LIN {X 0,Y 135.592,Z 571.454,A -85,B 0,C 180,E1 -25460.01,E2 -25460.01} C_VEL
LIN {X 0,Y 130.179,Z 578.331,A -85,B 0,C 180,E1 -25465.363,E2 -25465.363} C_VEL
LIN {X 0,Y 125.633,Z 584.379,A -85,B 0,C 180,E1 -25471.45,E2 -25471.45} C_VEL
LIN {X 0,Y 122.158,Z 589.423,A -85,B 0,C 180,E1 -25478.277,E2 -25478.277} C_VEL
LIN {X 0,Y 120.292,Z 592.378,A -85,B 0,C 180,E1 -25483.523,E2 -25483.523} C_VEL
LIN {X 0,Y 118.921,Z 595.269,A -85,B 0,C 180,E1 -25490.776,E2 -25490.776} C_VEL
LIN {X 0,Y 118.628,Z 597.068,A -85,B 0,C 180,E1 -25498.299,E2 -25498.299} C_VEL
LIN {X 0,Y 119.44,Z 597.753,A -85,B 0,C 180,E1 -25506.053,E2 -25506.053} C_VEL
LIN {X 0,Y 121.683,Z 597.158,A -85,B 0,C 180,E1 -25513.883,E2 -25513.883} C_VEL
LIN {X 0,Y 126.178,Z 595.007,A -85,B 0,C 180,E1 -25522.214,E2 -25522.214} C_VEL
LIN {X 0,Y 131.533,Z 591.96,A -85,B 0,C 180,E1 -25528.76,E2 -25528.76} C_VEL
LIN {X 0,Y 139.181,Z 587.216,A -85,B 0,C 180,E1 -25535.368,E2 -25535.368} C_VEL
LIN {X 0,Y 148.466,Z 580.898,A -85,B 0,C 180,E1 -25541.232,E2 -25541.232} C_VEL
LIN {X 0,Y 157.684,Z 573.958,A -85,B 0,C 180,E1 -25545.803,E2 -25545.803} C_VEL
LIN {X 0,Y 167.784,Z 565.497,A -85,B 0,C 180,E1 -25549.839,E2 -25549.839} C_VEL
LIN {X 0,Y 178,Z 555.977,A -85,B 0,C 180,E1 -25553.196,E2 -25553.196} C_VEL
LIN {X 0,Y 188.093,Z 545.484,A -85,B 0,C 180,E1 -25556.006,E2 -25556.006} C_VEL
LIN {X 0,Y 197.755,Z 534.153,A -85,B 0,C 180,E1 -25558.332,E2 -25558.332} C_VEL
LIN {X 0,Y 207.737,Z 520.677,A -85,B 0,C 180,E1 -25560.442,E2 -25560.442} C_VEL
LIN {X 0,Y 216.157,Z 507.546,A -85,B 0,C 180,E1 -25562.035,E2 -25562.035} C_VEL
LIN {X 0,Y 223.516,Z 494.335,A -85,B 0,C 180,E1 -25563.294,E2 -25563.294} C_VEL
LIN {X 0,Y 230.408,Z 479.829,A -85,B 0,C 180,E1 -25564.38,E2 -25564.38} C_VEL
LIN {X 0,Y 236.834,Z 463.137,A -85,B 0,C 180,E1 -25565.366,E2 -25565.366} C_VEL
LIN {X 0,Y 241.978,Z 445.87,A -85,B 0,C 180,E1 -25566.104,E2 -25566.104} C_VEL
LIN {X 0,Y 245.672,Z 428.764,A -85,B 0,C 180,E1 -25566.602,E2 -25566.602} C_VEL
LIN {X 0,Y 249.432,Z 401.164,A -85,B 0,C 180,E1 -25567.223,E2 -25567.223} C_VEL
LIN {X 0,Y 252.389,Z 377.643,A -85,B 0,C 180,E1 -25567.722,E2 -25567.722} C_VEL
LIN {X 0,Y 251.88,Z 375.905,A -85,B 0,C 180,E1 -25569.299,E2 -25569.299} C_VEL
LIN {X 0,Y 251.261,Z 374.694,A -85,B 0,C 180,E1 -25572.93,E2 -25572.93} C_VEL
LIN {X 0,Y 251.723,Z 376.03,A -85,B 0,C 180,E1 -25576.961,E2 -25576.961} C_VEL
LIN {X 0,Y 252.352,Z 378.18,A -85,B 0,C 180,E1 -25578.969,E2 -25578.969} C_VEL
LIN {X 0,Y 245.77,Z 429.103,A -85,B 0,C 180,E1 -25580.079,E2 -25580.079} C_VEL
LIN {X 0,Y 242.031,Z 446.842,A -85,B 0,C 180,E1 -25580.559,E2 -25580.559} C_VEL
LIN {X 0,Y 237.321,Z 462.811,A -85,B 0,C 180,E1 -25581.113,E2 -25581.113} C_VEL
LIN {X 0,Y 231.814,Z 477.633,A -85,B 0,C 180,E1 -25581.797,E2 -25581.797} C_VEL
LIN {X 0,Y 224.834,Z 493.11,A -85,B 0,C 180,E1 -25582.755,E2 -25582.755} C_VEL
LIN {X 0,Y 217.262,Z 507.328,A -85,B 0,C 180,E1 -25583.954,E2 -25583.954} C_VEL
LIN {X 0,Y 208.28,Z 521.6,A -85,B 0,C 180,E1 -25585.489,E2 -25585.489} C_VEL
LIN {X 0,Y 199.481,Z 533.795,A -85,B 0,C 180,E1 -25587.171,E2 -25587.171} C_VEL
LIN {X 0,Y 189.526,Z 546.009,A -85,B 0,C 180,E1 -25589.369,E2 -25589.369} C_VEL
LIN {X 0,Y 186.248,Z 549.75,A -85,B 0,C 180,E1 -25590.184,E2 -25590.184} C_VEL
LIN {X 0,Y 182.466,Z 553.642,A -85,B 0,C 180,E1 -25590.914,E2 -25590.914} C_VEL
LIN {X 0,Y 175.151,Z 559.9,A -85,B 0,C 180,E1 -25591.703,E2 -25591.703} C_VEL
LIN {X 0,Y 167.636,Z 565.745,A -85,B 0,C 180,E1 -25592.627,E2 -25592.627} C_VEL
LIN {X 0,Y 163.597,Z 568.989,A -85,B 0,C 180,E1 -25593.602,E2 -25593.602} C_VEL
LIN {X 0,Y 154.124,Z 576.822,A -85,B 0,C 180,E1 -25597.054,E2 -25597.054} C_VEL
LIN {X 0,Y 144.728,Z 583.846,A -85,B 0,C 180,E1 -25601.169,E2 -25601.169} C_VEL
LIN {X 0,Y 136.246,Z 589.755,A -85,B 0,C 180,E1 -25605.856,E2 -25605.856} C_VEL
LIN {X 0,Y 127.19,Z 595.559,A -85,B 0,C 180,E1 -25612.56,E2 -25612.56} C_VEL
LIN {X 0,Y 121.353,Z 599.067,A -85,B 0,C 180,E1 -25618.578,E2 -25618.578} C_VEL
LIN {X 0,Y 116.922,Z 601.669,A -85,B 0,C 180,E1 -25625.109,E2 -25625.109} C_VEL
LIN {X 0,Y 113.858,Z 603.302,A -85,B 0,C 180,E1 -25632.015,E2 -25632.015} C_VEL
LIN {X 0,Y 112.347,Z 604.045,A -85,B 0,C 180,E1 -25639.175,E2 -25639.175} C_VEL
LIN {X 0,Y 112.094,Z 603.844,A -85,B 0,C 180,E1 -25646.397,E2 -25646.397} C_VEL
LIN {X 0,Y 112.257,Z 603.413,A -85,B 0,C 180,E1 -25649.991,E2 -25649.991} C_VEL
LIN {X 0,Y 112.15,Z 602.645,A -85,B 0,C 180,E1 -25653.584,E2 -25653.584} C_VEL
LIN {X 0,Y 112.372,Z 600.386,A -85,B 0,C 180,E1 -25660.805,E2 -25660.805} C_VEL
LIN {X 0,Y 113.821,Z 597.066,A -85,B 0,C 180,E1 -25667.973,E2 -25667.973} C_VEL
LIN {X 0,Y 116.637,Z 592.573,A -85,B 0,C 180,E1 -25674.937,E2 -25674.937} C_VEL
LIN {X 0,Y 120.86,Z 586.935,A -85,B 0,C 180,E1 -25681.546,E2 -25681.546} C_VEL
LIN {X 0,Y 126.427,Z 579.919,A -85,B 0,C 180,E1 -25687.686,E2 -25687.686} C_VEL
LIN {X 0,Y 133.26,Z 571.437,A -85,B 0,C 180,E1 -25693.271,E2 -25693.271} C_VEL
LIN {X 0,Y 141.252,Z 561.3,A -85,B 0,C 180,E1 -25698.26,E2 -25698.26} C_VEL
LIN {X 0,Y 148.848,Z 550.863,A -85,B 0,C 180,E1 -25702.208,E2 -25702.208} C_VEL
LIN {X 0,Y 157.274,Z 538.45,A -85,B 0,C 180,E1 -25705.746,E2 -25705.746} C_VEL
LIN {X 0,Y 165.567,Z 524.865,A -85,B 0,C 180,E1 -25708.664,E2 -25708.664} C_VEL
LIN {X 0,Y 172.997,Z 510.8,A -85,B 0,C 180,E1 -25711.004,E2 -25711.004} C_VEL
LIN {X 0,Y 179.049,Z 497.991,A -85,B 0,C 180,E1 -25712.616,E2 -25712.616} C_VEL
LIN {X 0,Y 184.604,Z 484.152,A -85,B 0,C 180,E1 -25714.066,E2 -25714.066} C_VEL
LIN {X 0,Y 189.981,Z 468.245,A -85,B 0,C 180,E1 -25715.301,E2 -25715.301} C_VEL
LIN {X 0,Y 194.28,Z 452.182,A -85,B 0,C 180,E1 -25716.223,E2 -25716.223} C_VEL
LIN {X 0,Y 197.661,Z 435.216,A -85,B 0,C 180,E1 -25716.916,E2 -25716.916} C_VEL
LIN {X 0,Y 200.248,Z 413.846,A -85,B 0,C 180,E1 -25717.556,E2 -25717.556} C_VEL
LIN {X 0,Y 206.055,Z 356.958,A -85,B 0,C 180,E1 -25719.042,E2 -25719.042} C_VEL
LIN {X 0,Y 202.664,Z 348.652,A -85,B 0,C 180,E1 -25721.46,E2 -25721.46} C_VEL
LIN {X 0,Y 197.888,Z 339.554,A -85,B 0,C 180,E1 -25725.059,E2 -25725.059} C_VEL
LIN {X 0,Y 194.619,Z 333.664,A -85,B 0,C 180,E1 -25727.861,E2 -25727.861} C_VEL
LIN {X 0,Y 190.744,Z 326.828,A -85,B 0,C 180,E1 -25731.764,E2 -25731.764} C_VEL
LIN {X 0,Y 188.214,Z 322.78,A -85,B 0,C 180,E1 -25734.72,E2 -25734.72} C_VEL
LIN {X 0,Y 185.944,Z 318.938,A -85,B 0,C 180,E1 -25737.976,E2 -25737.976} C_VEL
LIN {X 0,Y 183.704,Z 314.93,A -85,B 0,C 180,E1 -25742.194,E2 -25742.194} C_VEL
LIN {X 0,Y 181.527,Z 311.165,A -85,B 0,C 180,E1 -25749.1,E2 -25749.1} C_VEL
LIN {X 0,Y 181.215,Z 310.726,A -85,B 0,C 180,E1 -25751.182,E2 -25751.182} C_VEL
LIN {X 0,Y 181.355,Z 311.109,A -85,B 0,C 180,E1 -25757.598,E2 -25757.598} C_VEL
LIN {X 0,Y 182.716,Z 314.596,A -85,B 0,C 180,E1 -25763.359,E2 -25763.359} C_VEL
LIN {X 0,Y 183.914,Z 315.929,A -85,B 0,C 180,E1 -25765.961,E2 -25765.961} C_VEL
LIN {X 0,Y 186.085,Z 319.594,A -85,B 0,C 180,E1 -25769.858,E2 -25769.858} C_VEL
LIN {X 0,Y 189.46,Z 325.124,A -85,B 0,C 180,E1 -25774.389,E2 -25774.389} C_VEL
LIN {X 0,Y 191.793,Z 328.987,A -85,B 0,C 180,E1 -25776.936,E2 -25776.936} C_VEL
LIN {X 0,Y 195.559,Z 335.364,A -85,B 0,C 180,E1 -25780.51,E2 -25780.51} C_VEL
LIN {X 0,Y 199.632,Z 342.86,A -85,B 0,C 180,E1 -25783.861,E2 -25783.861} C_VEL
LIN {X 0,Y 204.721,Z 352.73,A -85,B 0,C 180,E1 -25787.481,E2 -25787.481} C_VEL
LIN {X 0,Y 205.97,Z 355.322,A -85,B 0,C 180,E1 -25788.312,E2 -25788.312} C_VEL
LIN {X 0,Y 198.676,Z 425.073,A -85,B 0,C 180,E1 -25790.184,E2 -25790.184} C_VEL
LIN {X 0,Y 195.575,Z 442.344,A -85,B 0,C 180,E1 -25790.876,E2 -25790.876} C_VEL
LIN {X 0,Y 191.352,Z 459.391,A -85,B 0,C 180,E1 -25791.875,E2 -25791.875} C_VEL
LIN {X 0,Y 186.836,Z 473.785,A -85,B 0,C 180,E1 -25793.006,E2 -25793.006} C_VEL
LIN {X 0,Y 181.362,Z 488.387,A -85,B 0,C 180,E1 -25794.468,E2 -25794.468} C_VEL
LIN {X 0,Y 174.607,Z 503.527,A -85,B 0,C 180,E1 -25796.405,E2 -25796.405} C_VEL
LIN {X 0,Y 167.366,Z 517.429,A -85,B 0,C 180,E1 -25798.7,E2 -25798.7} C_VEL
LIN {X 0,Y 160.325,Z 529.42,A -85,B 0,C 180,E1 -25801.252,E2 -25801.252} C_VEL
LIN {X 0,Y 151.98,Z 542.111,A -85,B 0,C 180,E1 -25804.683,E2 -25804.683} C_VEL
LIN {X 0,Y 144.457,Z 552.67,A -85,B 0,C 180,E1 -25808.421,E2 -25808.421} C_VEL
LIN {X 0,Y 136.952,Z 562.378,A -85,B 0,C 180,E1 -25812.846,E2 -25812.846} C_VEL
LIN {X 0,Y 129.327,Z 571.783,A -85,B 0,C 180,E1 -25818.588,E2 -25818.588} C_VEL
LIN {X 0,Y 122.816,Z 579.635,A -85,B 0,C 180,E1 -25825.084,E2 -25825.084} C_VEL
LIN {X 0,Y 118.113,Z 585.569,A -85,B 0,C 180,E1 -25831.713,E2 -25831.713} C_VEL
LIN {X 0,Y 115.465,Z 589.228,A -85,B 0,C 180,E1 -25837,E2 -25837} C_VEL
LIN {X 0,Y 112.921,Z 593.101,A -85,B 0,C 180,E1 -25844.424,E2 -25844.424} C_VEL
LIN {X 0,Y 111.647,Z 595.89,A -85,B 0,C 180,E1 -25852.199,E2 -25852.199} C_VEL
LIN {X 0,Y 111.526,Z 597.161,A -85,B 0,C 180,E1 -25858.083,E2 -25858.083} C_VEL
LIN {X 0,Y 112.213,Z 597.912,A -85,B 0,C 180,E1 -25865.489,E2 -25865.489} C_VEL
LIN {X 0,Y 114.041,Z 597.7,A -85,B 0,C 180,E1 -25872.689,E2 -25872.689} C_VEL
LIN {X 0,Y 117.873,Z 596.291,A -85,B 0,C 180,E1 -25880.825,E2 -25880.825} C_VEL
LIN {X 0,Y 123.655,Z 593.462,A -85,B 0,C 180,E1 -25888.5,E2 -25888.5} C_VEL
LIN {X 0,Y 131.31,Z 589.2,A -85,B 0,C 180,E1 -25895.501,E2 -25895.501} C_VEL
LIN {X 0,Y 140.678,Z 583.443,A -85,B 0,C 180,E1 -25901.675,E2 -25901.675} C_VEL
LIN {X 0,Y 150.025,Z 577.049,A -85,B 0,C 180,E1 -25906.452,E2 -25906.452} C_VEL
LIN {X 0,Y 160.383,Z 569.194,A -85,B 0,C 180,E1 -25910.646,E2 -25910.646} C_VEL
LIN {X 0,Y 171.299,Z 559.856,A -85,B 0,C 180,E1 -25914.255,E2 -25914.255} C_VEL
LIN {X 0,Y 181.225,Z 550.299,A -85,B 0,C 180,E1 -25917.025,E2 -25917.025} C_VEL
LIN {X 0,Y 191.121,Z 539.644,A -85,B 0,C 180,E1 -25919.381,E2 -25919.381} C_VEL
LIN {X 0,Y 200.359,Z 528.42,A -85,B 0,C 180,E1 -25921.309,E2 -25921.309} C_VEL
LIN {X 0,Y 209.38,Z 515.849,A -85,B 0,C 180,E1 -25923.006,E2 -25923.006} C_VEL
LIN {X 0,Y 217.84,Z 502.246,A -85,B 0,C 180,E1 -25924.442,E2 -25924.442} C_VEL
LIN {X 0,Y 225.03,Z 488.838,A -85,B 0,C 180,E1 -25925.534,E2 -25925.534} C_VEL
LIN {X 0,Y 232.139,Z 472.857,A -85,B 0,C 180,E1 -25926.57,E2 -25926.57} C_VEL
LIN {X 0,Y 237.357,Z 458.347,A -85,B 0,C 180,E1 -25927.283,E2 -25927.283} C_VEL
LIN {X 0,Y 241.791,Z 442.785,A -85,B 0,C 180,E1 -25927.871,E2 -25927.871} C_VEL
LIN {X 0,Y 245.152,Z 426.835,A -85,B 0,C 180,E1 -25928.286,E2 -25928.286} C_VEL
LIN {X 0,Y 250.914,Z 383.242,A -85,B 0,C 180,E1 -25929.204,E2 -25929.204} C_VEL
LIN {X 0,Y 250.511,Z 382.29,A -85,B 0,C 180,E1 -25930.905,E2 -25930.905} C_VEL
LIN {X 0,Y 250.296,Z 381.743,A -85,B 0,C 180,E1 -25932.98,E2 -25932.98} C_VEL
LIN {X 0,Y 250.697,Z 383.034,A -85,B 0,C 180,E1 -25936.781,E2 -25936.781} C_VEL
LIN {X 0,Y 250.856,Z 383.838,A -85,B 0,C 180,E1 -25937.467,E2 -25937.467} C_VEL
LIN {X 0,Y 244.859,Z 429.052,A -85,B 0,C 180,E1 -25938.428,E2 -25938.428} C_VEL
LIN {X 0,Y 241.087,Z 446.514,A -85,B 0,C 180,E1 -25938.867,E2 -25938.867} C_VEL
LIN {X 0,Y 236.531,Z 461.763,A -85,B 0,C 180,E1 -25939.367,E2 -25939.367} C_VEL
LIN {X 0,Y 230.933,Z 476.71,A -85,B 0,C 180,E1 -25940.006,E2 -25940.006} C_VEL
LIN {X 0,Y 223.826,Z 492.289,A -85,B 0,C 180,E1 -25940.905,E2 -25940.905} C_VEL
LIN {X 0,Y 216.077,Z 506.592,A -85,B 0,C 180,E1 -25942.026,E2 -25942.026} C_VEL
LIN {X 0,Y 206.893,Z 520.947,A -85,B 0,C 180,E1 -25943.478,E2 -25943.478} C_VEL
LIN {X 0,Y 197.047,Z 534.196,A -85,B 0,C 180,E1 -25945.226,E2 -25945.226} C_VEL
LIN {X 0,Y 187.612,Z 545.401,A -85,B 0,C 180,E1 -25947.16,E2 -25947.16} C_VEL
LIN {X 0,Y 177.744,Z 555.928,A -85,B 0,C 180,E1 -25949.548,E2 -25949.548} C_VEL
LIN {X 0,Y 166.822,Z 566.161,A -85,B 0,C 180,E1 -25952.58,E2 -25952.58} C_VEL
LIN {X 0,Y 163.597,Z 568.989,A -85,B 0,C 180,E1 -25953.602,E2 -25953.602} C_VEL
LIN {X 0,Y 159.548,Z 572.171,A -85,B 0,C 180,E1 -25954.664,E2 -25954.664} C_VEL
LIN {X 0,Y 151.819,Z 577.208,A -85,B 0,C 180,E1 -25956.033,E2 -25956.033} C_VEL
LIN {X 0,Y 144.06,Z 581.798,A -85,B 0,C 180,E1 -25957.605,E2 -25957.605} C_VEL
LIN {X 0,Y 140.047,Z 584.247,A -85,B 0,C 180,E1 -25959.011,E2 -25959.011} C_VEL
LIN {X 0,Y 131.205,Z 589.978,A -85,B 0,C 180,E1 -25963.679,E2 -25963.679} C_VEL
LIN {X 0,Y 121.571,Z 595.694,A -85,B 0,C 180,E1 -25970.504,E2 -25970.504} C_VEL
LIN {X 0,Y 115.272,Z 599.087,A -85,B 0,C 180,E1 -25976.712,E2 -25976.712} C_VEL
LIN {X 0,Y 110.431,Z 601.637,A -85,B 0,C 180,E1 -25983.537,E2 -25983.537} C_VEL
LIN {X 0,Y 107.072,Z 603.168,A -85,B 0,C 180,E1 -25990.832,E2 -25990.832} C_VEL
LIN {X 0,Y 105.321,Z 603.861,A -85,B 0,C 180,E1 -25998.443,E2 -25998.443} C_VEL
LIN {X 0,Y 105.001,Z 603.568,A -85,B 0,C 180,E1 -26006.153,E2 -26006.153} C_VEL
LIN {X 0,Y 105.168,Z 603.103,A -85,B 0,C 180,E1 -26009.991,E2 -26009.991} C_VEL
LIN {X 0,Y 105.04,Z 602.323,A -85,B 0,C 180,E1 -26013.827,E2 -26013.827} C_VEL
LIN {X 0,Y 105.339,Z 599.966,A -85,B 0,C 180,E1 -26021.536,E2 -26021.536} C_VEL
LIN {X 0,Y 107.029,Z 596.596,A -85,B 0,C 180,E1 -26029.157,E2 -26029.157} C_VEL
LIN {X 0,Y 110.346,Z 591.711,A -85,B 0,C 180,E1 -26036.921,E2 -26036.921} C_VEL
LIN {X 0,Y 114.736,Z 586.244,A -85,B 0,C 180,E1 -26043.444,E2 -26043.444} C_VEL
LIN {X 0,Y 120.772,Z 579.17,A -85,B 0,C 180,E1 -26049.788,E2 -26049.788} C_VEL
LIN {X 0,Y 128.076,Z 570.56,A -85,B 0,C 180,E1 -26055.495,E2 -26055.495} C_VEL
LIN {X 0,Y 135.422,Z 561.672,A -85,B 0,C 180,E1 -26059.936,E2 -26059.936} C_VEL
LIN {X 0,Y 143.324,Z 551.33,A -85,B 0,C 180,E1 -26063.956,E2 -26063.956} C_VEL
LIN {X 0,Y 152.026,Z 539.037,A -85,B 0,C 180,E1 -26067.515,E2 -26067.515} C_VEL
LIN {X 0,Y 160.578,Z 525.567,A -85,B 0,C 180,E1 -26070.427,E2 -26070.427} C_VEL
LIN {X 0,Y 167.897,Z 512.3,A -85,B 0,C 180,E1 -26072.662,E2 -26072.662} C_VEL
LIN {X 0,Y 174.416,Z 499.109,A -85,B 0,C 180,E1 -26074.35,E2 -26074.35} C_VEL
LIN {X 0,Y 180.828,Z 483.59,A -85,B 0,C 180,E1 -26075.953,E2 -26075.953} C_VEL
LIN {X 0,Y 186.34,Z 467.641,A -85,B 0,C 180,E1 -26077.155,E2 -26077.155} C_VEL
LIN {X 0,Y 190.449,Z 452.593,A -85,B 0,C 180,E1 -26077.996,E2 -26077.996} C_VEL
LIN {X 0,Y 193.861,Z 436.047,A -85,B 0,C 180,E1 -26078.676,E2 -26078.676} C_VEL
LIN {X 0,Y 196.246,Z 417.895,A -85,B 0,C 180,E1 -26079.228,E2 -26079.228} C_VEL
LIN {X 0,Y 202.356,Z 360.051,A -85,B 0,C 180,E1 -26080.698,E2 -26080.698} C_VEL
LIN {X 0,Y 199.641,Z 353.521,A -85,B 0,C 180,E1 -26082.722,E2 -26082.722} C_VEL
LIN {X 0,Y 194.436,Z 343.102,A -85,B 0,C 180,E1 -26087.01,E2 -26087.01} C_VEL
LIN {X 0,Y 189.898,Z 334.931,A -85,B 0,C 180,E1 -26091.488,E2 -26091.488} C_VEL
LIN {X 0,Y 187.03,Z 329.885,A -85,B 0,C 180,E1 -26094.909,E2 -26094.909} C_VEL
LIN {X 0,Y 184.537,Z 325.617,A -85,B 0,C 180,E1 -26098.587,E2 -26098.587} C_VEL
LIN {X 0,Y 182.388,Z 321.658,A -85,B 0,C 180,E1 -26102.9,E2 -26102.9} C_VEL
LIN {X 0,Y 180.455,Z 317.888,A -85,B 0,C 180,E1 -26109.827,E2 -26109.827} C_VEL
LIN {X 0,Y 180.343,Z 318.059,A -85,B 0,C 180,E1 -26117.234,E2 -26117.234} C_VEL
LIN {X 0,Y 181.651,Z 321.579,A -85,B 0,C 180,E1 -26123.133,E2 -26123.133} C_VEL
LIN {X 0,Y 182.687,Z 322.781,A -85,B 0,C 180,E1 -26125.457,E2 -26125.457} C_VEL
LIN {X 0,Y 185.253,Z 327.269,A -85,B 0,C 180,E1 -26130.158,E2 -26130.158} C_VEL
LIN {X 0,Y 187.814,Z 331.646,A -85,B 0,C 180,E1 -26133.691,E2 -26133.691} C_VEL
LIN {X 0,Y 190.393,Z 336.056,A -85,B 0,C 180,E1 -26136.609,E2 -26136.609} C_VEL
LIN {X 0,Y 194.659,Z 343.675,A -85,B 0,C 180,E1 -26140.733,E2 -26140.733} C_VEL
LIN {X 0,Y 199.436,Z 353.112,A -85,B 0,C 180,E1 -26144.655,E2 -26144.655} C_VEL
LIN {X 0,Y 202.155,Z 358.635,A -85,B 0,C 180,E1 -26146.613,E2 -26146.613} C_VEL
LIN {X 0,Y 195.655,Z 420.719,A -85,B 0,C 180,E1 -26148.277,E2 -26148.277} C_VEL
LIN {X 0,Y 192.75,Z 438.379,A -85,B 0,C 180,E1 -26148.908,E2 -26148.908} C_VEL
LIN {X 0,Y 188.943,Z 454.628,A -85,B 0,C 180,E1 -26149.746,E2 -26149.746} C_VEL
LIN {X 0,Y 184.285,Z 470.153,A -85,B 0,C 180,E1 -26150.838,E2 -26150.838} C_VEL
LIN {X 0,Y 178.155,Z 486.634,A -85,B 0,C 180,E1 -26152.396,E2 -26152.396} C_VEL
LIN {X 0,Y 171.318,Z 501.736,A -85,B 0,C 180,E1 -26154.235,E2 -26154.235} C_VEL
LIN {X 0,Y 163.853,Z 515.919,A -85,B 0,C 180,E1 -26156.488,E2 -26156.488} C_VEL
LIN {X 0,Y 156.255,Z 528.585,A -85,B 0,C 180,E1 -26159.076,E2 -26159.076} C_VEL
LIN {X 0,Y 147.825,Z 541.122,A -85,B 0,C 180,E1 -26162.393,E2 -26162.393} C_VEL
LIN {X 0,Y 139.616,Z 552.238,A -85,B 0,C 180,E1 -26166.261,E2 -26166.261} C_VEL
LIN {X 0,Y 130.981,Z 562.946,A -85,B 0,C 180,E1 -26171.228,E2 -26171.228} C_VEL
LIN {X 0,Y 123.378,Z 571.846,A -85,B 0,C 180,E1 -26176.838,E2 -26176.838} C_VEL
LIN {X 0,Y 116.85,Z 579.247,A -85,B 0,C 180,E1 -26183.1,E2 -26183.1} C_VEL
LIN {X 0,Y 111.728,Z 585.314,A -85,B 0,C 180,E1 -26190.009,E2 -26190.009} C_VEL
LIN {X 0,Y 107.978,Z 590.184,A -85,B 0,C 180,E1 -26197.488,E2 -26197.488} C_VEL
LIN {X 0,Y 105.518,Z 593.832,A -85,B 0,C 180,E1 -26205.46,E2 -26205.46} C_VEL
LIN {X 0,Y 104.766,Z 595.399,A -85,B 0,C 180,E1 -26210.083,E2 -26210.083} C_VEL
LIN {X 0,Y 104.45,Z 597.408,A -85,B 0,C 180,E1 -26218.984,E2 -26218.984} C_VEL
LIN {X 0,Y 105.351,Z 598.141,A -85,B 0,C 180,E1 -26226.908,E2 -26226.908} C_VEL
LIN {X 0,Y 107.987,Z 597.76,A -85,B 0,C 180,E1 -26235.727,E2 -26235.727} C_VEL
LIN {X 0,Y 112.633,Z 596.11,A -85,B 0,C 180,E1 -26244.221,E2 -26244.221} C_VEL
LIN {X 0,Y 119.33,Z 593.114,A -85,B 0,C 180,E1 -26252.072,E2 -26252.072} C_VEL
LIN {X 0,Y 127.942,Z 588.655,A -85,B 0,C 180,E1 -26259.055,E2 -26259.055} C_VEL
LIN {X 0,Y 138.645,Z 582.369,A -85,B 0,C 180,E1 -26265.316,E2 -26265.316} C_VEL
LIN {X 0,Y 149.748,Z 574.959,A -85,B 0,C 180,E1 -26270.282,E2 -26270.282} C_VEL
LIN {X 0,Y 160.72,Z 566.677,A -85,B 0,C 180,E1 -26274.201,E2 -26274.201} C_VEL
LIN {X 0,Y 170.843,Z 558.141,A -85,B 0,C 180,E1 -26277.169,E2 -26277.169} C_VEL
LIN {X 0,Y 181.496,Z 548.045,A -85,B 0,C 180,E1 -26279.815,E2 -26279.815} C_VEL
LIN {X 0,Y 192.117,Z 536.535,A -85,B 0,C 180,E1 -26282.095,E2 -26282.095} C_VEL
LIN {X 0,Y 202.228,Z 523.982,A -85,B 0,C 180,E1 -26283.985,E2 -26283.985} C_VEL
LIN {X 0,Y 211.856,Z 510.148,A -85,B 0,C 180,E1 -26285.591,E2 -26285.591} C_VEL
LIN {X 0,Y 220.504,Z 495.62,A -85,B 0,C 180,E1 -26286.859,E2 -26286.859} C_VEL
LIN {X 0,Y 227.881,Z 480.857,A -85,B 0,C 180,E1 -26287.877,E2 -26287.877} C_VEL
LIN {X 0,Y 234.147,Z 465.432,A -85,B 0,C 180,E1 -26288.709,E2 -26288.709} C_VEL
LIN {X 0,Y 239.4,Z 449.103,A -85,B 0,C 180,E1 -26289.358,E2 -26289.358} C_VEL
LIN {X 0,Y 243.443,Z 432.16,A -85,B 0,C 180,E1 -26289.835,E2 -26289.835} C_VEL
LIN {X 0,Y 246.389,Z 413.634,A -85,B 0,C 180,E1 -26290.237,E2 -26290.237} C_VEL
LIN {X 0,Y 249.575,Z 389.433,A -85,B 0,C 180,E1 -26290.725,E2 -26290.725} C_VEL
LIN {X 0,Y 249.332,Z 388.783,A -85,B 0,C 180,E1 -26293.031,E2 -26293.031} C_VEL
LIN {X 0,Y 249.56,Z 389.655,A -85,B 0,C 180,E1 -26295.968,E2 -26295.968} C_VEL
LIN {X 0,Y 244.115,Z 429.219,A -85,B 0,C 180,E1 -26296.771,E2 -26296.771} C_VEL
LIN {X 0,Y 240.223,Z 446.862,A -85,B 0,C 180,E1 -26297.196,E2 -26297.196} C_VEL
LIN {X 0,Y 235.564,Z 462.083,A -85,B 0,C 180,E1 -26297.659,E2 -26297.659} C_VEL
LIN {X 0,Y 229.48,Z 477.855,A -85,B 0,C 180,E1 -26298.298,E2 -26298.298} C_VEL
LIN {X 0,Y 222.257,Z 493.146,A -85,B 0,C 180,E1 -26299.14,E2 -26299.14} C_VEL
LIN {X 0,Y 214.375,Z 507.243,A -85,B 0,C 180,E1 -26300.203,E2 -26300.203} C_VEL
LIN {X 0,Y 204.995,Z 521.426,A -85,B 0,C 180,E1 -26301.566,E2 -26301.566} C_VEL
LIN {X 0,Y 194.707,Z 534.846,A -85,B 0,C 180,E1 -26303.267,E2 -26303.267} C_VEL
LIN {X 0,Y 184.517,Z 546.454,A -85,B 0,C 180,E1 -26305.222,E2 -26305.222} C_VEL
LIN {X 0,Y 174.38,Z 556.766,A -85,B 0,C 180,E1 -26307.536,E2 -26307.536} C_VEL
LIN {X 0,Y 163.123,Z 566.855,A -85,B 0,C 180,E1 -26310.487,E2 -26310.487} C_VEL
LIN {X 0,Y 152.473,Z 575.372,A -85,B 0,C 180,E1 -26313.926,E2 -26313.926} C_VEL
LIN {X 0,Y 142.505,Z 582.602,A -85,B 0,C 180,E1 -26317.892,E2 -26317.892} C_VEL
LIN {X 0,Y 140.047,Z 584.247,A -85,B 0,C 180,E1 -26319.011,E2 -26319.011} C_VEL
LIN {X 0,Y 136.066,Z 586.648,A -85,B 0,C 180,E1 -26320.534,E2 -26320.534} C_VEL
LIN {X 0,Y 122.249,Z 592.933,A -85,B 0,C 180,E1 -26324.711,E2 -26324.711} C_VEL
LIN {X 0,Y 118.29,Z 594.673,A -85,B 0,C 180,E1 -26326.62,E2 -26326.62} C_VEL
LIN {X 0,Y 117.202,Z 595.212,A -85,B 0,C 180,E1 -26327.372,E2 -26327.372} C_VEL
LIN {X 0,Y 109.315,Z 599.127,A -85,B 0,C 180,E1 -26334.637,E2 -26334.637} C_VEL
LIN {X 0,Y 104.038,Z 601.57,A -85,B 0,C 180,E1 -26341.77,E2 -26341.77} C_VEL
LIN {X 0,Y 100.313,Z 603.035,A -85,B 0,C 180,E1 -26349.485,E2 -26349.485} C_VEL
LIN {X 0,Y 98.326,Z 603.671,A -85,B 0,C 180,E1 -26357.608,E2 -26357.608} C_VEL
LIN {X 0,Y 97.903,Z 603.287,A -85,B 0,C 180,E1 -26365.874,E2 -26365.874} C_VEL
LIN {X 0,Y 98.071,Z 602.776,A -85,B 0,C 180,E1 -26369.99,E2 -26369.99} C_VEL
LIN {X 0,Y 97.931,Z 601.996,A -85,B 0,C 180,E1 -26374.105,E2 -26374.105} C_VEL
LIN {X 0,Y 98.338,Z 599.543,A -85,B 0,C 180,E1 -26382.37,E2 -26382.37} C_VEL
LIN {X 0,Y 100.262,Z 596.093,A -85,B 0,C 180,E1 -26390.506,E2 -26390.506} C_VEL
LIN {X 0,Y 103.721,Z 591.415,A -85,B 0,C 180,E1 -26398.303,E2 -26398.303} C_VEL
LIN {X 0,Y 108.776,Z 585.547,A -85,B 0,C 180,E1 -26405.543,E2 -26405.543} C_VEL
LIN {X 0,Y 115.296,Z 578.387,A -85,B 0,C 180,E1 -26412.094,E2 -26412.094} C_VEL
LIN {X 0,Y 123.107,Z 569.664,A -85,B 0,C 180,E1 -26417.901,E2 -26417.901} C_VEL
LIN {X 0,Y 130.856,Z 560.62,A -85,B 0,C 180,E1 -26422.376,E2 -26422.376} C_VEL
LIN {X 0,Y 139.668,Z 549.454,A -85,B 0,C 180,E1 -26426.576,E2 -26426.576} C_VEL
LIN {X 0,Y 148.255,Z 537.632,A -85,B 0,C 180,E1 -26429.882,E2 -26429.882} C_VEL
LIN {X 0,Y 156.435,Z 525.104,A -85,B 0,C 180,E1 -26432.516,E2 -26432.516} C_VEL
LIN {X 0,Y 164.126,Z 511.508,A -85,B 0,C 180,E1 -26434.749,E2 -26434.749} C_VEL
LIN {X 0,Y 170.672,Z 498.504,A -85,B 0,C 180,E1 -26436.36,E2 -26436.36} C_VEL
LIN {X 0,Y 177.257,Z 482.878,A -85,B 0,C 180,E1 -26437.919,E2 -26437.919} C_VEL
LIN {X 0,Y 182.897,Z 466.832,A -85,B 0,C 180,E1 -26439.083,E2 -26439.083} C_VEL
LIN {X 0,Y 187.218,Z 451.196,A -85,B 0,C 180,E1 -26439.909,E2 -26439.909} C_VEL
LIN {X 0,Y 190.575,Z 434.853,A -85,B 0,C 180,E1 -26440.539,E2 -26440.539} C_VEL
LIN {X 0,Y 193.412,Z 412.301,A -85,B 0,C 180,E1 -26441.191,E2 -26441.191} C_VEL
LIN {X 0,Y 198.695,Z 363.055,A -85,B 0,C 180,E1 -26442.438,E2 -26442.438} C_VEL
LIN {X 0,Y 196.385,Z 357.593,A -85,B 0,C 180,E1 -26444.307,E2 -26444.307} C_VEL
LIN {X 0,Y 191.801,Z 348.326,A -85,B 0,C 180,E1 -26448.354,E2 -26448.354} C_VEL
LIN {X 0,Y 187.969,Z 341.08,A -85,B 0,C 180,E1 -26452.409,E2 -26452.409} C_VEL
LIN {X 0,Y 185.189,Z 336.029,A -85,B 0,C 180,E1 -26455.996,E2 -26455.996} C_VEL
LIN {X 0,Y 183.286,Z 332.501,A -85,B 0,C 180,E1 -26458.978,E2 -26458.978} C_VEL
LIN {X 0,Y 181.238,Z 328.568,A -85,B 0,C 180,E1 -26463.267,E2 -26463.267} C_VEL
LIN {X 0,Y 179.375,Z 324.847,A -85,B 0,C 180,E1 -26470.564,E2 -26470.564} C_VEL
LIN {X 0,Y 179.347,Z 325.085,A -85,B 0,C 180,E1 -26477.008,E2 -26477.008} C_VEL
LIN {X 0,Y 180.592,Z 328.536,A -85,B 0,C 180,E1 -26482.904,E2 -26482.904} C_VEL
LIN {X 0,Y 181.563,Z 329.838,A -85,B 0,C 180,E1 -26485.202,E2 -26485.202} C_VEL
LIN {X 0,Y 183.817,Z 333.934,A -85,B 0,C 180,E1 -26489.532,E2 -26489.532} C_VEL
LIN {X 0,Y 186.302,Z 338.369,A -85,B 0,C 180,E1 -26493.121,E2 -26493.121} C_VEL
LIN {X 0,Y 189.361,Z 343.776,A -85,B 0,C 180,E1 -26496.677,E2 -26496.677} C_VEL
LIN {X 0,Y 193.413,Z 351.546,A -85,B 0,C 180,E1 -26500.674,E2 -26500.674} C_VEL
LIN {X 0,Y 197.984,Z 360.981,A -85,B 0,C 180,E1 -26504.501,E2 -26504.501} C_VEL
LIN {X 0,Y 198.552,Z 362.263,A -85,B 0,C 180,E1 -26504.943,E2 -26504.943} C_VEL
LIN {X 0,Y 191.647,Z 425.034,A -85,B 0,C 180,E1 -26506.569,E2 -26506.569} C_VEL
LIN {X 0,Y 188.272,Z 443.015,A -85,B 0,C 180,E1 -26507.25,E2 -26507.25} C_VEL
LIN {X 0,Y 183.84,Z 459.988,A -85,B 0,C 180,E1 -26508.203,E2 -26508.203} C_VEL
LIN {X 0,Y 179.109,Z 474.326,A -85,B 0,C 180,E1 -26509.291,E2 -26509.291} C_VEL
LIN {X 0,Y 172.854,Z 490.009,A -85,B 0,C 180,E1 -26510.827,E2 -26510.827} C_VEL
LIN {X 0,Y 166.201,Z 504.032,A -85,B 0,C 180,E1 -26512.574,E2 -26512.574} C_VEL
LIN {X 0,Y 158.493,Z 517.946,A -85,B 0,C 180,E1 -26514.807,E2 -26514.807} C_VEL
LIN {X 0,Y 151.179,Z 529.599,A -85,B 0,C 180,E1 -26517.246,E2 -26517.246} C_VEL
LIN {X 0,Y 142.641,Z 541.765,A -85,B 0,C 180,E1 -26520.49,E2 -26520.49} C_VEL
LIN {X 0,Y 134.125,Z 552.81,A -85,B 0,C 180,E1 -26524.396,E2 -26524.396} C_VEL
LIN {X 0,Y 125.102,Z 563.469,A -85,B 0,C 180,E1 -26529.454,E2 -26529.454} C_VEL
LIN {X 0,Y 117.145,Z 572.336,A -85,B 0,C 180,E1 -26535.237,E2 -26535.237} C_VEL
LIN {X 0,Y 111.047,Z 578.837,A -85,B 0,C 180,E1 -26540.906,E2 -26540.906} C_VEL
LIN {X 0,Y 105.483,Z 585.027,A -85,B 0,C 180,E1 -26548.079,E2 -26548.079} C_VEL
LIN {X 0,Y 101.349,Z 589.972,A -85,B 0,C 180,E1 -26555.98,E2 -26555.98} C_VEL
LIN {X 0,Y 99.14,Z 592.949,A -85,B 0,C 180,E1 -26562.288,E2 -26562.288} C_VEL
LIN {X 0,Y 97.514,Z 595.865,A -85,B 0,C 180,E1 -26571.132,E2 -26571.132} C_VEL
LIN {X 0,Y 97.406,Z 597.691,A -85,B 0,C 180,E1 -26580.346,E2 -26580.346} C_VEL
LIN {X 0,Y 98.807,Z 598.401,A -85,B 0,C 180,E1 -26589.814,E2 -26589.814} C_VEL
LIN {X 0,Y 102.23,Z 597.821,A -85,B 0,C 180,E1 -26599.144,E2 -26599.144} C_VEL
LIN {X 0,Y 108.54,Z 595.68,A -85,B 0,C 180,E1 -26608.799,E2 -26608.799} C_VEL
LIN {X 0,Y 115.525,Z 592.7,A -85,B 0,C 180,E1 -26615.872,E2 -26615.872} C_VEL
LIN {X 0,Y 125.1,Z 588.022,A -85,B 0,C 180,E1 -26622.774,E2 -26622.774} C_VEL
LIN {X 0,Y 136.216,Z 581.823,A -85,B 0,C 180,E1 -26628.632,E2 -26628.632} C_VEL
LIN {X 0,Y 146.995,Z 574.936,A -85,B 0,C 180,E1 -26633.021,E2 -26633.021} C_VEL
LIN {X 0,Y 158.393,Z 566.67,A -85,B 0,C 180,E1 -26636.764,E2 -26636.764} C_VEL
LIN {X 0,Y 170.514,Z 556.699,A -85,B 0,C 180,E1 -26639.999,E2 -26639.999} C_VEL
LIN {X 0,Y 181.27,Z 546.629,A -85,B 0,C 180,E1 -26642.406,E2 -26642.406} C_VEL
LIN {X 0,Y 191.929,Z 535.236,A -85,B 0,C 180,E1 -26644.471,E2 -26644.471} C_VEL
LIN {X 0,Y 201.018,Z 524.12,A -85,B 0,C 180,E1 -26646.02,E2 -26646.02} C_VEL
LIN {X 0,Y 210.659,Z 510.614,A -85,B 0,C 180,E1 -26647.494,E2 -26647.494} C_VEL
LIN {X 0,Y 218.565,Z 497.772,A -85,B 0,C 180,E1 -26648.579,E2 -26648.579} C_VEL
LIN {X 0,Y 226.499,Z 482.381,A -85,B 0,C 180,E1 -26649.589,E2 -26649.589} C_VEL
LIN {X 0,Y 232.993,Z 467.057,A -85,B 0,C 180,E1 -26650.39,E2 -26650.39} C_VEL
LIN {X 0,Y 238.521,Z 450.633,A -85,B 0,C 180,E1 -26651.014,E2 -26651.014} C_VEL
LIN {X 0,Y 242.648,Z 434.282,A -85,B 0,C 180,E1 -26651.454,E2 -26651.454} C_VEL
LIN {X 0,Y 245.57,Z 417.245,A -85,B 0,C 180,E1 -26651.815,E2 -26651.815} C_VEL
LIN {X 0,Y 248.422,Z 395.959,A -85,B 0,C 180,E1 -26652.231,E2 -26652.231} C_VEL
LIN {X 0,Y 248.37,Z 396.032,A -85,B 0,C 180,E1 -26653.946,E2 -26653.946} C_VEL
LIN {X 0,Y 248.397,Z 396.198,A -85,B 0,C 180,E1 -26654.441,E2 -26654.441} C_VEL
LIN {X 0,Y 243.697,Z 429.284,A -85,B 0,C 180,E1 -26655.108,E2 -26655.108} C_VEL
LIN {X 0,Y 239.738,Z 446.81,A -85,B 0,C 180,E1 -26655.498,E2 -26655.498} C_VEL
LIN {X 0,Y 234.64,Z 463.053,A -85,B 0,C 180,E1 -26655.964,E2 -26655.964} C_VEL
LIN {X 0,Y 229.063,Z 477.142,A -85,B 0,C 180,E1 -26656.497,E2 -26656.497} C_VEL
LIN {X 0,Y 221.726,Z 492.508,A -85,B 0,C 180,E1 -26657.272,E2 -26657.272} C_VEL
LIN {X 0,Y 213.68,Z 506.697,A -85,B 0,C 180,E1 -26658.241,E2 -26658.241} C_VEL
LIN {X 0,Y 204.117,Z 520.916,A -85,B 0,C 180,E1 -26659.507,E2 -26659.507} C_VEL
LIN {X 0,Y 193.919,Z 533.943,A -85,B 0,C 180,E1 -26661.05,E2 -26661.05} C_VEL
LIN {X 0,Y 183.144,Z 545.951,A -85,B 0,C 180,E1 -26662.922,E2 -26662.922} C_VEL
LIN {X 0,Y 172.719,Z 556.308,A -85,B 0,C 180,E1 -26665.119,E2 -26665.119} C_VEL
LIN {X 0,Y 161.075,Z 566.386,A -85,B 0,C 180,E1 -26667.919,E2 -26667.919} C_VEL
LIN {X 0,Y 150.112,Z 574.807,A -85,B 0,C 180,E1 -26671.147,E2 -26671.147} C_VEL
LIN {X 0,Y 138.229,Z 582.99,A -85,B 0,C 180,E1 -26675.553,E2 -26675.553} C_VEL
LIN {X 0,Y 128.613,Z 588.925,A -85,B 0,C 180,E1 -26680.082,E2 -26680.082} C_VEL
LIN {X 0,Y 118.002,Z 594.796,A -85,B 0,C 180,E1 -26686.762,E2 -26686.762} C_VEL
LIN {X 0,Y 117.202,Z 595.212,A -85,B 0,C 180,E1 -26687.372,E2 -26687.372} C_VEL
LIN {X 0,Y 113.706,Z 596.754,A -85,B 0,C 180,E1 -26689.607,E2 -26689.607} C_VEL
LIN {X 0,Y 106.806,Z 598.987,A -85,B 0,C 180,E1 -26693.119,E2 -26693.119} C_VEL
LIN {X 0,Y 101.456,Z 600.447,A -85,B 0,C 180,E1 -26696.252,E2 -26696.252} C_VEL
LIN {X 0,Y 98.296,Z 601.342,A -85,B 0,C 180,E1 -26699.075,E2 -26699.075} C_VEL
LIN {X 0,Y 97.526,Z 601.575,A -85,B 0,C 180,E1 -26700.127,E2 -26700.127} C_VEL
LIN {X 0,Y 93.624,Z 602.906,A -85,B 0,C 180,E1 -26707.945,E2 -26707.945} C_VEL
LIN {X 0,Y 91.346,Z 603.443,A -85,B 0,C 180,E1 -26716.645,E2 -26716.645} C_VEL
LIN {X 0,Y 90.797,Z 603.004,A -85,B 0,C 180,E1 -26725.55,E2 -26725.55} C_VEL
LIN {X 0,Y 90.968,Z 602.443,A -85,B 0,C 180,E1 -26729.989,E2 -26729.989} C_VEL
LIN {X 0,Y 90.819,Z 601.628,A -85,B 0,C 180,E1 -26734.427,E2 -26734.427} C_VEL
LIN {X 0,Y 91.354,Z 599.103,A -85,B 0,C 180,E1 -26743.332,E2 -26743.332} C_VEL
LIN {X 0,Y 93.568,Z 595.542,A -85,B 0,C 180,E1 -26752.047,E2 -26752.047} C_VEL
LIN {X 0,Y 97.418,Z 590.803,A -85,B 0,C 180,E1 -26760.318,E2 -26760.318} C_VEL
LIN {X 0,Y 102.972,Z 584.814,A -85,B 0,C 180,E1 -26767.885,E2 -26767.885} C_VEL
LIN {X 0,Y 110.03,Z 577.522,A -85,B 0,C 180,E1 -26774.622,E2 -26774.622} C_VEL
LIN {X 0,Y 118.351,Z 568.719,A -85,B 0,C 180,E1 -26780.516,E2 -26780.516} C_VEL
LIN {X 0,Y 127.757,Z 558.125,A -85,B 0,C 180,E1 -26785.588,E2 -26785.588} C_VEL
LIN {X 0,Y 136.58,Z 547.227,A -85,B 0,C 180,E1 -26789.415,E2 -26789.415} C_VEL
LIN {X 0,Y 145.445,Z 535.151,A -85,B 0,C 180,E1 -26792.591,E2 -26792.591} C_VEL
LIN {X 0,Y 153.208,Z 523.437,A -85,B 0,C 180,E1 -26794.936,E2 -26794.936} C_VEL
LIN {X 0,Y 161.17,Z 509.617,A -85,B 0,C 180,E1 -26797.078,E2 -26797.078} C_VEL
LIN {X 0,Y 167.147,Z 497.845,A -85,B 0,C 180,E1 -26798.458,E2 -26798.458} C_VEL
LIN {X 0,Y 173.9,Z 482.106,A -85,B 0,C 180,E1 -26799.966,E2 -26799.966} C_VEL
LIN {X 0,Y 179.663,Z 465.894,A -85,B 0,C 180,E1 -26801.09,E2 -26801.09} C_VEL
LIN {X 0,Y 183.942,Z 450.643,A -85,B 0,C 180,E1 -26801.858,E2 -26801.858} C_VEL
LIN {X 0,Y 187.254,Z 434.833,A -85,B 0,C 180,E1 -26802.437,E2 -26802.437} C_VEL
LIN {X 0,Y 190.045,Z 413.426,A -85,B 0,C 180,E1 -26803.045,E2 -26803.045} C_VEL
LIN {X 0,Y 195.253,Z 366.422,A -85,B 0,C 180,E1 -26804.19,E2 -26804.19} C_VEL
LIN {X 0,Y 192.154,Z 359.522,A -85,B 0,C 180,E1 -26806.913,E2 -26806.913} C_VEL
LIN {X 0,Y 188.928,Z 352.74,A -85,B 0,C 180,E1 -26810.12,E2 -26810.12} C_VEL
LIN {X 0,Y 185.357,Z 345.744,A -85,B 0,C 180,E1 -26814.302,E2 -26814.302} C_VEL
LIN {X 0,Y 183.219,Z 341.795,A -85,B 0,C 180,E1 -26817.372,E2 -26817.372} C_VEL
LIN {X 0,Y 181.699,Z 338.829,A -85,B 0,C 180,E1 -26820.001,E2 -26820.001} C_VEL
LIN {X 0,Y 180.009,Z 335.369,A -85,B 0,C 180,E1 -26823.851,E2 -26823.851} C_VEL
LIN {X 0,Y 178.466,Z 332.005,A -85,B 0,C 180,E1 -26830.144,E2 -26830.144} C_VEL
LIN {X 0,Y 178.279,Z 332,A -85,B 0,C 180,E1 -26836.02,E2 -26836.02} C_VEL
LIN {X 0,Y 178.405,Z 332.604,A -85,B 0,C 180,E1 -26837.522,E2 -26837.522} C_VEL
LIN {X 0,Y 179.663,Z 335.68,A -85,B 0,C 180,E1 -26843.029,E2 -26843.029} C_VEL
LIN {X 0,Y 180.339,Z 336.674,A -85,B 0,C 180,E1 -26844.698,E2 -26844.698} C_VEL
LIN {X 0,Y 182.46,Z 340.729,A -85,B 0,C 180,E1 -26848.998,E2 -26848.998} C_VEL
LIN {X 0,Y 184.8,Z 345.038,A -85,B 0,C 180,E1 -26852.525,E2 -26852.525} C_VEL
LIN {X 0,Y 187.69,Z 350.503,A -85,B 0,C 180,E1 -26856.081,E2 -26856.081} C_VEL
LIN {X 0,Y 191.293,Z 357.667,A -85,B 0,C 180,E1 -26859.807,E2 -26859.807} C_VEL
LIN {X 0,Y 195.022,Z 365.747,A -85,B 0,C 180,E1 -26863.129,E2 -26863.129} C_VEL
LIN {X 0,Y 189.706,Z 414.735,A -85,B 0,C 180,E1 -26864.393,E2 -26864.393} C_VEL
LIN {X 0,Y 187.214,Z 431.86,A -85,B 0,C 180,E1 -26864.891,E2 -26864.891} C_VEL
LIN {X 0,Y 183.594,Z 448.532,A -85,B 0,C 180,E1 -26865.598,E2 -26865.598} C_VEL
LIN {X 0,Y 178.908,Z 464.837,A -85,B 0,C 180,E1 -26866.581,E2 -26866.581} C_VEL
LIN {X 0,Y 173.676,Z 479.444,A -85,B 0,C 180,E1 -26867.73,E2 -26867.73} C_VEL
LIN {X 0,Y 166.606,Z 495.634,A -85,B 0,C 180,E1 -26869.405,E2 -26869.405} C_VEL
LIN {X 0,Y 159.053,Z 510.159,A -85,B 0,C 180,E1 -26871.391,E2 -26871.391} C_VEL
LIN {X 0,Y 151.225,Z 523.12,A -85,B 0,C 180,E1 -26873.672,E2 -26873.672} C_VEL
LIN {X 0,Y 142.377,Z 536.042,A -85,B 0,C 180,E1 -26876.642,E2 -26876.642} C_VEL
LIN {X 0,Y 133.779,Z 547.308,A -85,B 0,C 180,E1 -26880.071,E2 -26880.071} C_VEL
LIN {X 0,Y 124.571,Z 558.23,A -85,B 0,C 180,E1 -26884.517,E2 -26884.517} C_VEL
LIN {X 0,Y 115.07,Z 568.582,A -85,B 0,C 180,E1 -26890.381,E2 -26890.381} C_VEL
LIN {X 0,Y 107.183,Z 576.63,A -85,B 0,C 180,E1 -26896.742,E2 -26896.742} C_VEL
LIN {X 0,Y 100.759,Z 583.23,A -85,B 0,C 180,E1 -26904.004,E2 -26904.004} C_VEL
LIN {X 0,Y 95.788,Z 588.605,A -85,B 0,C 180,E1 -26912.112,E2 -26912.112} C_VEL
LIN {X 0,Y 92.7,Z 592.278,A -85,B 0,C 180,E1 -26919.726,E2 -26919.726} C_VEL
LIN {X 0,Y 90.778,Z 595.206,A -85,B 0,C 180,E1 -26928.05,E2 -26928.05} C_VEL
LIN {X 0,Y 90.179,Z 597.421,A -85,B 0,C 180,E1 -26937.89,E2 -26937.89} C_VEL
LIN {X 0,Y 91.271,Z 598.484,A -85,B 0,C 180,E1 -26948.037,E2 -26948.037} C_VEL
LIN {X 0,Y 94.413,Z 598.372,A -85,B 0,C 180,E1 -26958.12,E2 -26958.12} C_VEL
LIN {X 0,Y 99.907,Z 596.993,A -85,B 0,C 180,E1 -26967.595,E2 -26967.595} C_VEL
LIN {X 0,Y 107.624,Z 594.204,A -85,B 0,C 180,E1 -26976.112,E2 -26976.112} C_VEL
LIN {X 0,Y 117.335,Z 590.031,A -85,B 0,C 180,E1 -26983.426,E2 -26983.426} C_VEL
LIN {X 0,Y 128.655,Z 584.375,A -85,B 0,C 180,E1 -26989.538,E2 -26989.538} C_VEL
LIN {X 0,Y 140.018,Z 577.836,A -85,B 0,C 180,E1 -26994.237,E2 -26994.237} C_VEL
LIN {X 0,Y 151.569,Z 570.246,A -85,B 0,C 180,E1 -26998.021,E2 -26998.021} C_VEL
LIN {X 0,Y 163.447,Z 561.266,A -85,B 0,C 180,E1 -27001.194,E2 -27001.194} C_VEL
LIN {X 0,Y 174.299,Z 551.977,A -85,B 0,C 180,E1 -27003.611,E2 -27003.611} C_VEL
LIN {X 0,Y 185.263,Z 541.386,A -85,B 0,C 180,E1 -27005.674,E2 -27005.674} C_VEL
LIN {X 0,Y 195.806,Z 529.582,A -85,B 0,C 180,E1 -27007.439,E2 -27007.439} C_VEL
LIN {X 0,Y 205.449,Z 517.151,A -85,B 0,C 180,E1 -27008.857,E2 -27008.857} C_VEL
LIN {X 0,Y 214.092,Z 504.38,A -85,B 0,C 180,E1 -27009.986,E2 -27009.986} C_VEL
LIN {X 0,Y 222.681,Z 489.419,A -85,B 0,C 180,E1 -27011.004,E2 -27011.004} C_VEL
LIN {X 0,Y 229.78,Z 474.379,A -85,B 0,C 180,E1 -27011.825,E2 -27011.825} C_VEL
LIN {X 0,Y 235.672,Z 458.97,A -85,B 0,C 180,E1 -27012.444,E2 -27012.444} C_VEL
LIN {X 0,Y 240.174,Z 444.037,A -85,B 0,C 180,E1 -27012.913,E2 -27012.913} C_VEL
LIN {X 0,Y 243.78,Z 427.873,A -85,B 0,C 180,E1 -27013.257,E2 -27013.257} C_VEL
LIN {X 0,Y 244.219,Z 425.152,A -85,B 0,C 180,E1 -27013.309,E2 -27013.309} C_VEL
LIN {X 0,Y 241.057,Z 440.577,A -85,B 0,C 180,E1 -27013.672,E2 -27013.672} C_VEL
LIN {X 0,Y 236.779,Z 455.875,A -85,B 0,C 180,E1 -27014.011,E2 -27014.011} C_VEL
LIN {X 0,Y 230.534,Z 472.854,A -85,B 0,C 180,E1 -27014.543,E2 -27014.543} C_VEL
LIN {X 0,Y 223.9,Z 487.235,A -85,B 0,C 180,E1 -27015.149,E2 -27015.149} C_VEL
LIN {X 0,Y 216.509,Z 500.788,A -85,B 0,C 180,E1 -27015.912,E2 -27015.912} C_VEL
LIN {X 0,Y 207.581,Z 514.776,A -85,B 0,C 180,E1 -27016.963,E2 -27016.963} C_VEL
LIN {X 0,Y 197.911,Z 527.721,A -85,B 0,C 180,E1 -27018.201,E2 -27018.201} C_VEL
LIN {X 0,Y 188.05,Z 539.236,A -85,B 0,C 180,E1 -27019.654,E2 -27019.654} C_VEL
LIN {X 0,Y 177.454,Z 550.164,A -85,B 0,C 180,E1 -27021.445,E2 -27021.445} C_VEL
LIN {X 0,Y 165.296,Z 561.123,A -85,B 0,C 180,E1 -27023.908,E2 -27023.908} C_VEL
LIN {X 0,Y 153.511,Z 570.413,A -85,B 0,C 180,E1 -27026.77,E2 -27026.77} C_VEL
LIN {X 0,Y 142.281,Z 578.303,A -85,B 0,C 180,E1 -27030.175,E2 -27030.175} C_VEL
LIN {X 0,Y 131.615,Z 584.967,A -85,B 0,C 180,E1 -27034.13,E2 -27034.13} C_VEL
LIN {X 0,Y 121.75,Z 590.458,A -85,B 0,C 180,E1 -27038.795,E2 -27038.795} C_VEL
LIN {X 0,Y 114.966,Z 593.909,A -85,B 0,C 180,E1 -27042.803,E2 -27042.803} C_VEL
LIN {X 0,Y 106.996,Z 597.685,A -85,B 0,C 180,E1 -27048.93,E2 -27048.93} C_VEL
LIN {X 0,Y 98.001,Z 601.413,A -85,B 0,C 180,E1 -27059.376,E2 -27059.376} C_VEL
LIN {X 0,Y 97.526,Z 601.575,A -85,B 0,C 180,E1 -27060.127,E2 -27060.127} C_VEL
LIN {X 0,Y 95.011,Z 602.278,A -85,B 0,C 180,E1 -27063.287,E2 -27063.287} C_VEL
LIN {X 0,Y 89.775,Z 603.012,A -85,B 0,C 180,E1 -27068.495,E2 -27068.495} C_VEL
LIN {X 0,Y 85.984,Z 603.217,A -85,B 0,C 180,E1 -27073.063,E2 -27073.063} C_VEL
LIN {X 0,Y 84.243,Z 603.187,A -85,B 0,C 180,E1 -27076.882,E2 -27076.882} C_VEL
LIN {X 0,Y 83.998,Z 603.155,A -85,B 0,C 180,E1 -27078.218,E2 -27078.218} C_VEL
LIN {X 0,Y 83.715,Z 602.721,A -85,B 0,C 180,E1 -27085.173,E2 -27085.173} C_VEL
LIN {X 0,Y 83.872,Z 602.111,A -85,B 0,C 180,E1 -27089.988,E2 -27089.988} C_VEL
LIN {X 0,Y 83.733,Z 601.243,A -85,B 0,C 180,E1 -27094.803,E2 -27094.803} C_VEL
LIN {X 0,Y 84.383,Z 598.662,A -85,B 0,C 180,E1 -27104.457,E2 -27104.457} C_VEL
LIN {X 0,Y 87.856,Z 593.898,A -85,B 0,C 180,E1 -27116.088,E2 -27116.088} C_VEL
LIN {X 0,Y 92.645,Z 588.76,A -85,B 0,C 180,E1 -27124.663,E2 -27124.663} C_VEL
LIN {X 0,Y 99.131,Z 582.405,A -85,B 0,C 180,E1 -27132.324,E2 -27132.324} C_VEL
LIN {X 0,Y 107.831,Z 573.871,A -85,B 0,C 180,E1 -27139.498,E2 -27139.498} C_VEL
LIN {X 0,Y 117.518,Z 563.92,A -85,B 0,C 180,E1 -27145.298,E2 -27145.298} C_VEL
LIN {X 0,Y 126.399,Z 553.947,A -85,B 0,C 180,E1 -27149.503,E2 -27149.503} C_VEL
LIN {X 0,Y 135.893,Z 542.279,A -85,B 0,C 180,E1 -27153.12,E2 -27153.12} C_VEL
LIN {X 0,Y 145.188,Z 529.56,A -85,B 0,C 180,E1 -27155.996,E2 -27155.996} C_VEL
LIN {X 0,Y 153.615,Z 516.243,A -85,B 0,C 180,E1 -27158.324,E2 -27158.324} C_VEL
LIN {X 0,Y 161.576,Z 501.868,A -85,B 0,C 180,E1 -27160.131,E2 -27160.131} C_VEL
LIN {X 0,Y 168.452,Z 486.963,A -85,B 0,C 180,E1 -27161.625,E2 -27161.625} C_VEL
LIN {X 0,Y 174.683,Z 470.775,A -85,B 0,C 180,E1 -27162.822,E2 -27162.822} C_VEL
LIN {X 0,Y 179.627,Z 454.802,A -85,B 0,C 180,E1 -27163.671,E2 -27163.671} C_VEL
LIN {X 0,Y 183.382,Z 438.897,A -85,B 0,C 180,E1 -27164.289,E2 -27164.289} C_VEL
LIN {X 0,Y 186.063,Z 421.748,A -85,B 0,C 180,E1 -27164.78,E2 -27164.78} C_VEL
LIN {X 0,Y 191.887,Z 369.78,A -85,B 0,C 180,E1 -27166.06,E2 -27166.06} C_VEL
LIN {X 0,Y 187.711,Z 360.435,A -85,B 0,C 180,E1 -27170.209,E2 -27170.209} C_VEL
LIN {X 0,Y 183.989,Z 352.659,A -85,B 0,C 180,E1 -27174.711,E2 -27174.711} C_VEL
LIN {X 0,Y 181.628,Z 348.154,A -85,B 0,C 180,E1 -27178.258,E2 -27178.258} C_VEL
LIN {X 0,Y 180.383,Z 345.566,A -85,B 0,C 180,E1 -27180.596,E2 -27180.596} C_VEL
LIN {X 0,Y 178.852,Z 342.243,A -85,B 0,C 180,E1 -27184.298,E2 -27184.298} C_VEL
LIN {X 0,Y 177.403,Z 338.916,A -85,B 0,C 180,E1 -27190.913,E2 -27190.913} C_VEL
LIN {X 0,Y 177.364,Z 339.156,A -85,B 0,C 180,E1 -27196.572,E2 -27196.572} C_VEL
LIN {X 0,Y 178.463,Z 342.499,A -85,B 0,C 180,E1 -27202.406,E2 -27202.406} C_VEL
LIN {X 0,Y 179.185,Z 343.63,A -85,B 0,C 180,E1 -27204.329,E2 -27204.329} C_VEL
LIN {X 0,Y 181.075,Z 347.407,A -85,B 0,C 180,E1 -27208.371,E2 -27208.371} C_VEL
LIN {X 0,Y 183.597,Z 352.254,A -85,B 0,C 180,E1 -27212.323,E2 -27212.323} C_VEL
LIN {X 0,Y 186.762,Z 358.614,A -85,B 0,C 180,E1 -27216.289,E2 -27216.289} C_VEL
LIN {X 0,Y 189.819,Z 365.191,A -85,B 0,C 180,E1 -27219.531,E2 -27219.531} C_VEL
LIN {X 0,Y 191.739,Z 369.688,A -85,B 0,C 180,E1 -27221.362,E2 -27221.362} C_VEL
LIN {X 0,Y 185.188,Z 425.775,A -85,B 0,C 180,E1 -27222.726,E2 -27222.726} C_VEL
LIN {X 0,Y 181.769,Z 443.205,A -85,B 0,C 180,E1 -27223.343,E2 -27223.343} C_VEL
LIN {X 0,Y 177.144,Z 460.224,A -85,B 0,C 180,E1 -27224.235,E2 -27224.235} C_VEL
LIN {X 0,Y 172.175,Z 474.611,A -85,B 0,C 180,E1 -27225.251,E2 -27225.251} C_VEL
LIN {X 0,Y 165.361,Z 490.828,A -85,B 0,C 180,E1 -27226.749,E2 -27226.749} C_VEL
LIN {X 0,Y 157.849,Z 505.687,A -85,B 0,C 180,E1 -27228.536,E2 -27228.536} C_VEL
LIN {X 0,Y 149.73,Z 519.441,A -85,B 0,C 180,E1 -27230.69,E2 -27230.69} C_VEL
LIN {X 0,Y 141.162,Z 532.09,A -85,B 0,C 180,E1 -27233.324,E2 -27233.324} C_VEL
LIN {X 0,Y 132.811,Z 542.977,A -85,B 0,C 180,E1 -27236.256,E2 -27236.256} C_VEL
LIN {X 0,Y 123.632,Z 553.891,A -85,B 0,C 180,E1 -27240.182,E2 -27240.182} C_VEL
LIN {X 0,Y 114.982,Z 563.248,A -85,B 0,C 180,E1 -27244.679,E2 -27244.679} C_VEL
LIN {X 0,Y 105.995,Z 572.215,A -85,B 0,C 180,E1 -27250.649,E2 -27250.649} C_VEL
LIN {X 0,Y 98.224,Z 579.659,A -85,B 0,C 180,E1 -27257.615,E2 -27257.615} C_VEL
LIN {X 0,Y 91.573,Z 586.111,A -85,B 0,C 180,E1 -27266.165,E2 -27266.165} C_VEL
LIN {X 0,Y 87.272,Z 590.671,A -85,B 0,C 180,E1 -27274.63,E2 -27274.63} C_VEL
LIN {X 0,Y 84.23,Z 594.365,A -85,B 0,C 180,E1 -27284.507,E2 -27284.507} C_VEL
LIN {X 0,Y 83.241,Z 596.301,A -85,B 0,C 180,E1 -27291.756,E2 -27291.756} C_VEL
LIN {X 0,Y 83.341,Z 598.117,A -85,B 0,C 180,E1 -27302.507,E2 -27302.507} C_VEL
LIN {X 0,Y 84.983,Z 598.796,A -85,B 0,C 180,E1 -27311.898,E2 -27311.898} C_VEL
LIN {X 0,Y 88.963,Z 598.441,A -85,B 0,C 180,E1 -27322.2,E2 -27322.2} C_VEL
LIN {X 0,Y 95.556,Z 596.846,A -85,B 0,C 180,E1 -27331.972,E2 -27331.972} C_VEL
LIN {X 0,Y 104.415,Z 593.925,A -85,B 0,C 180,E1 -27340.466,E2 -27340.466} C_VEL
LIN {X 0,Y 115.161,Z 589.527,A -85,B 0,C 180,E1 -27347.567,E2 -27347.567} C_VEL
LIN {X 0,Y 128.086,Z 583.277,A -85,B 0,C 180,E1 -27353.698,E2 -27353.698} C_VEL
LIN {X 0,Y 140.644,Z 576.137,A -85,B 0,C 180,E1 -27358.154,E2 -27358.154} C_VEL
LIN {X 0,Y 152.931,Z 568.058,A -85,B 0,C 180,E1 -27361.625,E2 -27361.625} C_VEL
LIN {X 0,Y 165.177,Z 558.862,A -85,B 0,C 180,E1 -27364.436,E2 -27364.436} C_VEL
LIN {X 0,Y 176.913,Z 548.712,A -85,B 0,C 180,E1 -27366.686,E2 -27366.686} C_VEL
LIN {X 0,Y 188.41,Z 537.201,A -85,B 0,C 180,E1 -27368.58,E2 -27368.58} C_VEL
LIN {X 0,Y 198.42,Z 525.756,A -85,B 0,C 180,E1 -27370.006,E2 -27370.006} C_VEL
LIN {X 0,Y 207.794,Z 513.477,A -85,B 0,C 180,E1 -27371.223,E2 -27371.223} C_VEL
LIN {X 0,Y 217.365,Z 498.667,A -85,B 0,C 180,E1 -27372.316,E2 -27372.316} C_VEL
LIN {X 0,Y 223.595,Z 487.312,A -85,B 0,C 180,E1 -27372.987,E2 -27372.987} C_VEL
LIN {X 0,Y 223.877,Z 486.771,A -85,B 0,C 180,E1 -27373.295,E2 -27373.295} C_VEL
LIN {X 0,Y 216.384,Z 500.381,A -85,B 0,C 180,E1 -27373.986,E2 -27373.986} C_VEL
LIN {X 0,Y 207.32,Z 514.408,A -85,B 0,C 180,E1 -27374.945,E2 -27374.945} C_VEL
LIN {X 0,Y 198.295,Z 526.304,A -85,B 0,C 180,E1 -27375.968,E2 -27375.968} C_VEL
LIN {X 0,Y 187.757,Z 538.463,A -85,B 0,C 180,E1 -27377.343,E2 -27377.343} C_VEL
LIN {X 0,Y 176.586,Z 549.778,A -85,B 0,C 180,E1 -27379.04,E2 -27379.04} C_VEL
LIN {X 0,Y 164.126,Z 560.736,A -85,B 0,C 180,E1 -27381.343,E2 -27381.343} C_VEL
LIN {X 0,Y 151.95,Z 570.014,A -85,B 0,C 180,E1 -27383.999,E2 -27383.999} C_VEL
LIN {X 0,Y 141.682,Z 577.049,A -85,B 0,C 180,E1 -27386.753,E2 -27386.753} C_VEL
LIN {X 0,Y 127.745,Z 585.374,A -85,B 0,C 180,E1 -27391.477,E2 -27391.477} C_VEL
LIN {X 0,Y 114.936,Z 591.946,A -85,B 0,C 180,E1 -27397.342,E2 -27397.342} C_VEL
LIN {X 0,Y 105.814,Z 596.028,A -85,B 0,C 180,E1 -27403.052,E2 -27403.052} C_VEL
LIN {X 0,Y 97.938,Z 599.225,A -85,B 0,C 180,E1 -27409.76,E2 -27409.76} C_VEL
LIN {X 0,Y 89.085,Z 602.242,A -85,B 0,C 180,E1 -27421.737,E2 -27421.737} C_VEL
LIN {X 0,Y 85.403,Z 603.088,A -85,B 0,C 180,E1 -27430.77,E2 -27430.77} C_VEL
LIN {X 0,Y 83.998,Z 603.155,A -85,B 0,C 180,E1 -27438.218,E2 -27438.218} C_VEL
LIN {X 0,Y 82.979,Z 602.957,A -85,B 0,C 180,E1 -27442.204,E2 -27442.204} C_VEL
LIN {X 0,Y 81.199,Z 602.524,A -85,B 0,C 180,E1 -27446.157,E2 -27446.157} C_VEL
LIN {X 0,Y 76.873,Z 600.407,A -85,B 0,C 180,E1 -27457.348,E2 -27457.348} C_VEL
LIN {X 0,Y 76.806,Z 599.723,A -85,B 0,C 180,E1 -27460.321,E2 -27460.321} C_VEL
LIN {X 0,Y 78.639,Z 596.441,A -85,B 0,C 180,E1 -27470.932,E2 -27470.932} C_VEL
LIN {X 0,Y 82.611,Z 592.117,A -85,B 0,C 180,E1 -27480.678,E2 -27480.678} C_VEL
LIN {X 0,Y 88.419,Z 586.595,A -85,B 0,C 180,E1 -27489.469,E2 -27489.469} C_VEL
LIN {X 0,Y 95.939,Z 579.711,A -85,B 0,C 180,E1 -27497.083,E2 -27497.083} C_VEL
LIN {X 0,Y 104.828,Z 571.405,A -85,B 0,C 180,E1 -27503.545,E2 -27503.545} C_VEL
LIN {X 0,Y 113.549,Z 562.844,A -85,B 0,C 180,E1 -27508.306,E2 -27508.306} C_VEL
LIN {X 0,Y 122.54,Z 553.038,A -85,B 0,C 180,E1 -27512.312,E2 -27512.312} C_VEL
LIN {X 0,Y 132.765,Z 540.809,A -85,B 0,C 180,E1 -27515.92,E2 -27515.92} C_VEL
LIN {X 0,Y 142.392,Z 527.84,A -85,B 0,C 180,E1 -27518.663,E2 -27518.663} C_VEL
LIN {X 0,Y 151.178,Z 514.028,A -85,B 0,C 180,E1 -27520.918,E2 -27520.918} C_VEL
LIN {X 0,Y 159.26,Z 499.572,A -85,B 0,C 180,E1 -27522.583,E2 -27522.583} C_VEL
LIN {X 0,Y 166.305,Z 484.271,A -85,B 0,C 180,E1 -27524.001,E2 -27524.001} C_VEL
LIN {X 0,Y 172.294,Z 468.578,A -85,B 0,C 180,E1 -27525.037,E2 -27525.037} C_VEL
LIN {X 0,Y 176.717,Z 454.17,A -85,B 0,C 180,E1 -27525.755,E2 -27525.755} C_VEL
LIN {X 0,Y 180.36,Z 439.047,A -85,B 0,C 180,E1 -27526.312,E2 -27526.312} C_VEL
LIN {X 0,Y 183.072,Z 422.238,A -85,B 0,C 180,E1 -27526.769,E2 -27526.769} C_VEL
LIN {X 0,Y 188.699,Z 373.553,A -85,B 0,C 180,E1 -27527.913,E2 -27527.913} C_VEL
LIN {X 0,Y 185.254,Z 365.463,A -85,B 0,C 180,E1 -27531.701,E2 -27531.701} C_VEL
LIN {X 0,Y 182.138,Z 358.664,A -85,B 0,C 180,E1 -27535.835,E2 -27535.835} C_VEL
LIN {X 0,Y 179.448,Z 352.943,A -85,B 0,C 180,E1 -27540.45,E2 -27540.45} C_VEL
LIN {X 0,Y 177.673,Z 349.069,A -85,B 0,C 180,E1 -27544.847,E2 -27544.847} C_VEL
LIN {X 0,Y 176.434,Z 345.948,A -85,B 0,C 180,E1 -27550.974,E2 -27550.974} C_VEL
LIN {X 0,Y 176.379,Z 346.224,A -85,B 0,C 180,E1 -27556.413,E2 -27556.413} C_VEL
LIN {X 0,Y 177.446,Z 349.528,A -85,B 0,C 180,E1 -27562.278,E2 -27562.278} C_VEL
LIN {X 0,Y 178.045,Z 350.596,A -85,B 0,C 180,E1 -27563.972,E2 -27563.972} C_VEL
LIN {X 0,Y 179.831,Z 354.363,A -85,B 0,C 180,E1 -27567.969,E2 -27567.969} C_VEL
LIN {X 0,Y 182.154,Z 359.018,A -85,B 0,C 180,E1 -27571.768,E2 -27571.768} C_VEL
LIN {X 0,Y 185.22,Z 365.557,A -85,B 0,C 180,E1 -27575.813,E2 -27575.813} C_VEL
LIN {X 0,Y 188.17,Z 372.313,A -85,B 0,C 180,E1 -27579.072,E2 -27579.072} C_VEL
LIN {X 0,Y 188.51,Z 373.038,A -85,B 0,C 180,E1 -27579.412,E2 -27579.412} C_VEL
LIN {X 0,Y 187.958,Z 378.604,A -85,B 0,C 180,E1 -27579.609,E2 -27579.609} C_VEL
LIN {X 0,Y 182.255,Z 425.902,A -85,B 0,C 180,E1 -27580.711,E2 -27580.711} C_VEL
LIN {X 0,Y 178.812,Z 443.141,A -85,B 0,C 180,E1 -27581.291,E2 -27581.291} C_VEL
LIN {X 0,Y 174.134,Z 460.11,A -85,B 0,C 180,E1 -27582.142,E2 -27582.142} C_VEL
LIN {X 0,Y 168.661,Z 475.572,A -85,B 0,C 180,E1 -27583.19,E2 -27583.19} C_VEL
LIN {X 0,Y 161.68,Z 491.645,A -85,B 0,C 180,E1 -27584.629,E2 -27584.629} C_VEL
LIN {X 0,Y 153.959,Z 506.442,A -85,B 0,C 180,E1 -27586.364,E2 -27586.364} C_VEL
LIN {X 0,Y 145.649,Z 520.061,A -85,B 0,C 180,E1 -27588.445,E2 -27588.445} C_VEL
LIN {X 0,Y 136.825,Z 532.674,A -85,B 0,C 180,E1 -27591.018,E2 -27591.018} C_VEL
LIN {X 0,Y 128.199,Z 543.499,A -85,B 0,C 180,E1 -27593.902,E2 -27593.902} C_VEL
LIN {X 0,Y 118.665,Z 554.361,A -85,B 0,C 180,E1 -27597.801,E2 -27597.801} C_VEL
LIN {X 0,Y 109.737,Z 563.571,A -85,B 0,C 180,E1 -27602.241,E2 -27602.241} C_VEL
LIN {X 0,Y 100.192,Z 572.621,A -85,B 0,C 180,E1 -27608.403,E2 -27608.403} C_VEL
LIN {X 0,Y 92.896,Z 579.182,A -85,B 0,C 180,E1 -27614.657,E2 -27614.657} C_VEL
LIN {X 0,Y 86.07,Z 585.375,A -85,B 0,C 180,E1 -27622.838,E2 -27622.838} C_VEL
LIN {X 0,Y 80.777,Z 590.418,A -85,B 0,C 180,E1 -27632.505,E2 -27632.505} C_VEL
LIN {X 0,Y 78.012,Z 593.444,A -85,B 0,C 180,E1 -27640.392,E2 -27640.392} C_VEL
LIN {X 0,Y 76.07,Z 596.58,A -85,B 0,C 180,E1 -27652.491,E2 -27652.491} C_VEL
LIN {X 0,Y 76.371,Z 598.345,A -85,B 0,C 180,E1 -27664.079,E2 -27664.079} C_VEL
LIN {X 0,Y 78.798,Z 599.058,A -85,B 0,C 180,E1 -27675.537,E2 -27675.537} C_VEL
LIN {X 0,Y 83.989,Z 598.517,A -85,B 0,C 180,E1 -27686.819,E2 -27686.819} C_VEL
LIN {X 0,Y 92.852,Z 596.42,A -85,B 0,C 180,E1 -27697.76,E2 -27697.76} C_VEL
LIN {X 0,Y 101.837,Z 593.547,A -85,B 0,C 180,E1 -27705.084,E2 -27705.084} C_VEL
LIN {X 0,Y 113.62,Z 589.009,A -85,B 0,C 180,E1 -27711.806,E2 -27711.806} C_VEL
LIN {X 0,Y 126.66,Z 582.941,A -85,B 0,C 180,E1 -27717.269,E2 -27717.269} C_VEL
LIN {X 0,Y 140.629,Z 575.215,A -85,B 0,C 180,E1 -27721.643,E2 -27721.643} C_VEL
LIN {X 0,Y 153.38,Z 566.937,A -85,B 0,C 180,E1 -27724.781,E2 -27724.781} C_VEL
LIN {X 0,Y 165.742,Z 557.675,A -85,B 0,C 180,E1 -27727.307,E2 -27727.307} C_VEL
LIN {X 0,Y 178.083,Z 547.074,A -85,B 0,C 180,E1 -27729.364,E2 -27729.364} C_VEL
LIN {X 0,Y 189.033,Z 536.226,A -85,B 0,C 180,E1 -27730.948,E2 -27730.948} C_VEL
LIN {X 0,Y 199.611,Z 524.074,A -85,B 0,C 180,E1 -27732.291,E2 -27732.291} C_VEL
LIN {X 0,Y 204.122,Z 518.315,A -85,B 0,C 180,E1 -27732.834,E2 -27732.834} C_VEL
LIN {X 0,Y 203.47,Z 519.216,A -85,B 0,C 180,E1 -27733.294,E2 -27733.294} C_VEL
LIN {X 0,Y 194.031,Z 530.87,A -85,B 0,C 180,E1 -27734.312,E2 -27734.312} C_VEL
LIN {X 0,Y 184.118,Z 541.617,A -85,B 0,C 180,E1 -27735.521,E2 -27735.521} C_VEL
LIN {X 0,Y 172.821,Z 552.29,A -85,B 0,C 180,E1 -27737.114,E2 -27737.114} C_VEL
LIN {X 0,Y 160.103,Z 562.826,A -85,B 0,C 180,E1 -27739.292,E2 -27739.292} C_VEL
LIN {X 0,Y 147.678,Z 571.83,A -85,B 0,C 180,E1 -27741.862,E2 -27741.862} C_VEL
LIN {X 0,Y 135.685,Z 579.347,A -85,B 0,C 180,E1 -27744.97,E2 -27744.97} C_VEL
LIN {X 0,Y 124.17,Z 585.735,A -85,B 0,C 180,E1 -27748.67,E2 -27748.67} C_VEL
LIN {X 0,Y 113.326,Z 591.005,A -85,B 0,C 180,E1 -27753.141,E2 -27753.141} C_VEL
LIN {X 0,Y 105.753,Z 594.302,A -85,B 0,C 180,E1 -27757.098,E2 -27757.098} C_VEL
LIN {X 0,Y 92.553,Z 599.265,A -85,B 0,C 180,E1 -27766.877,E2 -27766.877} C_VEL
LIN {X 0,Y 85.088,Z 601.516,A -85,B 0,C 180,E1 -27775.683,E2 -27775.683} C_VEL
LIN {X 0,Y 80.517,Z 602.656,A -85,B 0,C 180,E1 -27784.111,E2 -27784.111} C_VEL
LIN {X 0,Y 76.937,Z 602.877,A -85,B 0,C 180,E1 -27797.853,E2 -27797.853} C_VEL
LIN {X 0,Y 76.608,Z 602.431,A -85,B 0,C 180,E1 -27804.724,E2 -27804.724} C_VEL
LIN {X 0,Y 76.768,Z 601.766,A -85,B 0,C 180,E1 -27809.987,E2 -27809.987} C_VEL
LIN {X 0,Y 76.806,Z 599.723,A -85,B 0,C 180,E1 -27820.321,E2 -27820.321} C_VEL
LIN {X 0,Y 76.694,Z 598.623,A -85,B 0,C 180,E1 -27824.649,E2 -27824.649} C_VEL
LIN {X 0,Y 75.406,Z 596.31,A -85,B 0,C 180,E1 -27831.857,E2 -27831.857} C_VEL
LIN {X 0,Y 74.93,Z 594.077,A -85,B 0,C 180,E1 -27837.713,E2 -27837.713} C_VEL
LIN {X 0,Y 75.787,Z 592.214,A -85,B 0,C 180,E1 -27841.969,E2 -27841.969} C_VEL
LIN {X 0,Y 76.41,Z 591.543,A -85,B 0,C 180,E1 -27843.301,E2 -27843.301} C_VEL
LIN {X 0,Y 82.956,Z 585.863,A -85,B 0,C 180,E1 -27852.651,E2 -27852.651} C_VEL
LIN {X 0,Y 91.149,Z 578.861,A -85,B 0,C 180,E1 -27860.428,E2 -27860.428} C_VEL
LIN {X 0,Y 100.697,Z 570.407,A -85,B 0,C 180,E1 -27866.858,E2 -27866.858} C_VEL
LIN {X 0,Y 111.284,Z 560.291,A -85,B 0,C 180,E1 -27872.124,E2 -27872.124} C_VEL
LIN {X 0,Y 121.124,Z 549.792,A -85,B 0,C 180,E1 -27876.038,E2 -27876.038} C_VEL
LIN {X 0,Y 131.479,Z 537.488,A -85,B 0,C 180,E1 -27879.271,E2 -27879.271} C_VEL
LIN {X 0,Y 140.68,Z 525.018,A -85,B 0,C 180,E1 -27881.628,E2 -27881.628} C_VEL
LIN {X 0,Y 149.184,Z 511.662,A -85,B 0,C 180,E1 -27883.583,E2 -27883.583} C_VEL
LIN {X 0,Y 157.227,Z 497.117,A -85,B 0,C 180,E1 -27885.124,E2 -27885.124} C_VEL
LIN {X 0,Y 164.448,Z 481.333,A -85,B 0,C 180,E1 -27886.439,E2 -27886.439} C_VEL
LIN {X 0,Y 170.559,Z 465.063,A -85,B 0,C 180,E1 -27887.401,E2 -27887.401} C_VEL
LIN {X 0,Y 175.293,Z 449.052,A -85,B 0,C 180,E1 -27888.065,E2 -27888.065} C_VEL
LIN {X 0,Y 178.781,Z 432.684,A -85,B 0,C 180,E1 -27888.578,E2 -27888.578} C_VEL
LIN {X 0,Y 181.902,Z 409.329,A -85,B 0,C 180,E1 -27889.145,E2 -27889.145} C_VEL
LIN {X 0,Y 185.673,Z 377.348,A -85,B 0,C 180,E1 -27889.866,E2 -27889.866} C_VEL
LIN {X 0,Y 183.111,Z 371.1,A -85,B 0,C 180,E1 -27892.934,E2 -27892.934} C_VEL
LIN {X 0,Y 180.442,Z 364.871,A -85,B 0,C 180,E1 -27896.804,E2 -27896.804} C_VEL
LIN {X 0,Y 178.068,Z 359.504,A -85,B 0,C 180,E1 -27901.235,E2 -27901.235} C_VEL
LIN {X 0,Y 176.485,Z 355.842,A -85,B 0,C 180,E1 -27905.488,E2 -27905.488} C_VEL
LIN {X 0,Y 175.418,Z 352.904,A -85,B 0,C 180,E1 -27911.557,E2 -27911.557} C_VEL
LIN {X 0,Y 175.394,Z 353.337,A -85,B 0,C 180,E1 -27916.291,E2 -27916.291} C_VEL
LIN {X 0,Y 176.418,Z 356.541,A -85,B 0,C 180,E1 -27922.111,E2 -27922.111} C_VEL
LIN {X 0,Y 176.934,Z 357.639,A -85,B 0,C 180,E1 -27923.682,E2 -27923.682} C_VEL
LIN {X 0,Y 178.534,Z 361.15,A -85,B 0,C 180,E1 -27927.434,E2 -27927.434} C_VEL
LIN {X 0,Y 180.823,Z 365.955,A -85,B 0,C 180,E1 -27931.359,E2 -27931.359} C_VEL
LIN {X 0,Y 183.717,Z 372.637,A -85,B 0,C 180,E1 -27935.372,E2 -27935.372} C_VEL
LIN {X 0,Y 185.534,Z 376.969,A -85,B 0,C 180,E1 -27937.495,E2 -27937.495} C_VEL
LIN {X 0,Y 179.623,Z 425.661,A -85,B 0,C 180,E1 -27938.631,E2 -27938.631} C_VEL
LIN {X 0,Y 176.166,Z 442.775,A -85,B 0,C 180,E1 -27939.166,E2 -27939.166} C_VEL
LIN {X 0,Y 171.764,Z 458.7,A -85,B 0,C 180,E1 -27939.91,E2 -27939.91} C_VEL
LIN {X 0,Y 166.17,Z 474.528,A -85,B 0,C 180,E1 -27940.898,E2 -27940.898} C_VEL
LIN {X 0,Y 159.839,Z 489.218,A -85,B 0,C 180,E1 -27942.111,E2 -27942.111} C_VEL
LIN {X 0,Y 152.469,Z 503.461,A -85,B 0,C 180,E1 -27943.603,E2 -27943.603} C_VEL
LIN {X 0,Y 144.115,Z 517.187,A -85,B 0,C 180,E1 -27945.503,E2 -27945.503} C_VEL
LIN {X 0,Y 134.958,Z 530.248,A -85,B 0,C 180,E1 -27947.908,E2 -27947.908} C_VEL
LIN {X 0,Y 125.26,Z 542.338,A -85,B 0,C 180,E1 -27950.872,E2 -27950.872} C_VEL
LIN {X 0,Y 115.289,Z 553.429,A -85,B 0,C 180,E1 -27954.623,E2 -27954.623} C_VEL
LIN {X 0,Y 105.773,Z 562.867,A -85,B 0,C 180,E1 -27959.018,E2 -27959.018} C_VEL
LIN {X 0,Y 96.923,Z 570.919,A -85,B 0,C 180,E1 -27964.223,E2 -27964.223} C_VEL
LIN {X 0,Y 87.837,Z 578.703,A -85,B 0,C 180,E1 -27971.347,E2 -27971.347} C_VEL
LIN {X 0,Y 80.243,Z 585.084,A -85,B 0,C 180,E1 -27979.924,E2 -27979.924} C_VEL
LIN {X 0,Y 74.426,Z 590.163,A -85,B 0,C 180,E1 -27990.013,E2 -27990.013} C_VEL
LIN {X 0,Y 70.492,Z 594.143,A -85,B 0,C 180,E1 -28001.515,E2 -28001.515} C_VEL
LIN {X 0,Y 68.856,Z 597.003,A -85,B 0,C 180,E1 -28014.111,E2 -28014.111} C_VEL
LIN {X 0,Y 69.453,Z 598.567,A -85,B 0,C 180,E1 -28025.945,E2 -28025.945} C_VEL
LIN {X 0,Y 71.941,Z 599.231,A -85,B 0,C 180,E1 -28036.852,E2 -28036.852} C_VEL
LIN {X 0,Y 76.033,Z 599.071,A -85,B 0,C 180,E1 -28046.314,E2 -28046.314} C_VEL
LIN {X 0,Y 83.894,Z 597.738,A -85,B 0,C 180,E1 -28057.169,E2 -28057.169} C_VEL
LIN {X 0,Y 95.798,Z 594.575,A -85,B 0,C 180,E1 -28067.283,E2 -28067.283} C_VEL
LIN {X 0,Y 109.413,Z 589.797,A -85,B 0,C 180,E1 -28074.71,E2 -28074.71} C_VEL
LIN {X 0,Y 122.9,Z 583.932,A -85,B 0,C 180,E1 -28079.998,E2 -28079.998} C_VEL
LIN {X 0,Y 137.427,Z 576.381,A -85,B 0,C 180,E1 -28084.203,E2 -28084.203} C_VEL
LIN {X 0,Y 151.277,Z 567.827,A -85,B 0,C 180,E1 -28087.325,E2 -28087.325} C_VEL
LIN {X 0,Y 164.871,Z 558.029,A -85,B 0,C 180,E1 -28089.816,E2 -28089.816} C_VEL
LIN {X 0,Y 177.396,Z 547.532,A -85,B 0,C 180,E1 -28091.685,E2 -28091.685} C_VEL
LIN {X 0,Y 185.493,Z 539.789,A -85,B 0,C 180,E1 -28092.755,E2 -28092.755} C_VEL
LIN {X 0,Y 184.855,Z 540.458,A -85,B 0,C 180,E1 -28093.116,E2 -28093.116} C_VEL
LIN {X 0,Y 172.525,Z 552.001,A -85,B 0,C 180,E1 -28094.638,E2 -28094.638} C_VEL
LIN {X 0,Y 159.545,Z 562.515,A -85,B 0,C 180,E1 -28096.633,E2 -28096.633} C_VEL
LIN {X 0,Y 146.778,Z 571.494,A -85,B 0,C 180,E1 -28098.96,E2 -28098.96} C_VEL
LIN {X 0,Y 135.873,Z 578.158,A -85,B 0,C 180,E1 -28101.388,E2 -28101.388} C_VEL
LIN {X 0,Y 123.83,Z 584.72,A -85,B 0,C 180,E1 -28104.744,E2 -28104.744} C_VEL
LIN {X 0,Y 109.571,Z 591.297,A -85,B 0,C 180,E1 -28110,E2 -28110} C_VEL
LIN {X 0,Y 101.595,Z 594.513,A -85,B 0,C 180,E1 -28113.876,E2 -28113.876} C_VEL
LIN {X 0,Y 91.826,Z 597.89,A -85,B 0,C 180,E1 -28120.047,E2 -28120.047} C_VEL
LIN {X 0,Y 83.454,Z 600.426,A -85,B 0,C 180,E1 -28127.632,E2 -28127.632} C_VEL
LIN {X 0,Y 76.729,Z 601.999,A -85,B 0,C 180,E1 -28136.649,E2 -28136.649} C_VEL
LIN {X 0,Y 72.017,Z 602.729,A -85,B 0,C 180,E1 -28147.01,E2 -28147.01} C_VEL
LIN {X 0,Y 69.782,Z 602.545,A -85,B 0,C 180,E1 -28158.366,E2 -28158.366} C_VEL
LIN {X 0,Y 69.518,Z 602.141,A -85,B 0,C 180,E1 -28164.184,E2 -28164.184} C_VEL
LIN {X 0,Y 69.686,Z 601.424,A -85,B 0,C 180,E1 -28169.986,E2 -28169.986} C_VEL
LIN {X 0,Y 69.796,Z 599.217,A -85,B 0,C 180,E1 -28181.603,E2 -28181.603} C_VEL
LIN {X 0,Y 71.99,Z 595.922,A -85,B 0,C 180,E1 -28192.97,E2 -28192.97} C_VEL
LIN {X 0,Y 76.41,Z 591.543,A -85,B 0,C 180,E1 -28203.301,E2 -28203.301} C_VEL
LIN {X 0,Y 78.065,Z 589.56,A -85,B 0,C 180,E1 -28207.222,E2 -28207.222} C_VEL
LIN {X 0,Y 79.82,Z 585.924,A -85,B 0,C 180,E1 -28213.797,E2 -28213.797} C_VEL
LIN {X 0,Y 82.411,Z 581.89,A -85,B 0,C 180,E1 -28219.948,E2 -28219.948} C_VEL
LIN {X 0,Y 85.232,Z 579.158,A -85,B 0,C 180,E1 -28223.009,E2 -28223.009} C_VEL
LIN {X 0,Y 95.584,Z 570.54,A -85,B 0,C 180,E1 -28229.736,E2 -28229.736} C_VEL
LIN {X 0,Y 106.644,Z 560.49,A -85,B 0,C 180,E1 -28234.952,E2 -28234.952} C_VEL
LIN {X 0,Y 116.498,Z 550.459,A -85,B 0,C 180,E1 -28238.659,E2 -28238.659} C_VEL
LIN {X 0,Y 127.537,Z 537.826,A -85,B 0,C 180,E1 -28241.878,E2 -28241.878} C_VEL
LIN {X 0,Y 136.975,Z 525.432,A -85,B 0,C 180,E1 -28244.128,E2 -28244.128} C_VEL
LIN {X 0,Y 145.869,Z 511.885,A -85,B 0,C 180,E1 -28246.022,E2 -28246.022} C_VEL
LIN {X 0,Y 153.894,Z 497.819,A -85,B 0,C 180,E1 -28247.422,E2 -28247.422} C_VEL
LIN {X 0,Y 161.254,Z 482.245,A -85,B 0,C 180,E1 -28248.662,E2 -28248.662} C_VEL
LIN {X 0,Y 167.471,Z 466.275,A -85,B 0,C 180,E1 -28249.554,E2 -28249.554} C_VEL
LIN {X 0,Y 172.003,Z 451.439,A -85,B 0,C 180,E1 -28250.159,E2 -28250.159} C_VEL
LIN {X 0,Y 175.923,Z 434.404,A -85,B 0,C 180,E1 -28250.662,E2 -28250.662} C_VEL
LIN {X 0,Y 178.904,Z 413.784,A -85,B 0,C 180,E1 -28251.152,E2 -28251.152} C_VEL
LIN {X 0,Y 182.814,Z 381.153,A -85,B 0,C 180,E1 -28251.865,E2 -28251.865} C_VEL
LIN {X 0,Y 180.181,Z 374.415,A -85,B 0,C 180,E1 -28255.527,E2 -28255.527} C_VEL
LIN {X 0,Y 177.976,Z 369.226,A -85,B 0,C 180,E1 -28259.235,E2 -28259.235} C_VEL
LIN {X 0,Y 176.454,Z 365.547,A -85,B 0,C 180,E1 -28262.641,E2 -28262.641} C_VEL
LIN {X 0,Y 175.35,Z 362.703,A -85,B 0,C 180,E1 -28266.015,E2 -28266.015} C_VEL
LIN {X 0,Y 174.454,Z 359.918,A -85,B 0,C 180,E1 -28271.622,E2 -28271.622} C_VEL
LIN {X 0,Y 174.409,Z 360.346,A -85,B 0,C 180,E1 -28276.023,E2 -28276.023} C_VEL
LIN {X 0,Y 175.391,Z 363.548,A -85,B 0,C 180,E1 -28281.942,E2 -28281.942} C_VEL
LIN {X 0,Y 177.093,Z 367.555,A -85,B 0,C 180,E1 -28286.531,E2 -28286.531} C_VEL
LIN {X 0,Y 179.285,Z 372.527,A -85,B 0,C 180,E1 -28290.639,E2 -28290.639} C_VEL
LIN {X 0,Y 182.23,Z 379.702,A -85,B 0,C 180,E1 -28294.926,E2 -28294.926} C_VEL
LIN {X 0,Y 182.686,Z 380.842,A -85,B 0,C 180,E1 -28295.506,E2 -28295.506} C_VEL
LIN {X 0,Y 177.169,Z 425.345,A -85,B 0,C 180,E1 -28296.499,E2 -28296.499} C_VEL
LIN {X 0,Y 173.728,Z 442.279,A -85,B 0,C 180,E1 -28296.981,E2 -28296.981} C_VEL
LIN {X 0,Y 169.243,Z 458.398,A -85,B 0,C 180,E1 -28297.678,E2 -28297.678} C_VEL
LIN {X 0,Y 163.133,Z 475.346,A -85,B 0,C 180,E1 -28298.674,E2 -28298.674} C_VEL
LIN {X 0,Y 155.855,Z 491.537,A -85,B 0,C 180,E1 -28299.964,E2 -28299.964} C_VEL
LIN {X 0,Y 147.796,Z 506.378,A -85,B 0,C 180,E1 -28301.513,E2 -28301.513} C_VEL
LIN {X 0,Y 139.002,Z 520.131,A -85,B 0,C 180,E1 -28303.393,E2 -28303.393} C_VEL
LIN {X 0,Y 128.94,Z 533.686,A -85,B 0,C 180,E1 -28305.935,E2 -28305.935} C_VEL
LIN {X 0,Y 118.186,Z 546.185,A -85,B 0,C 180,E1 -28309.16,E2 -28309.16} C_VEL
LIN {X 0,Y 107.984,Z 556.671,A -85,B 0,C 180,E1 -28312.998,E2 -28312.998} C_VEL
LIN {X 0,Y 98.207,Z 565.686,A -85,B 0,C 180,E1 -28317.552,E2 -28317.552} C_VEL
LIN {X 0,Y 87.872,Z 574.401,A -85,B 0,C 180,E1 -28323.917,E2 -28323.917} C_VEL
LIN {X 0,Y 78.755,Z 581.592,A -85,B 0,C 180,E1 -28331.814,E2 -28331.814} C_VEL
LIN {X 0,Y 70.994,Z 587.613,A -85,B 0,C 180,E1 -28341.889,E2 -28341.889} C_VEL
LIN {X 0,Y 65.702,Z 592.087,A -85,B 0,C 180,E1 -28353.081,E2 -28353.081} C_VEL
LIN {X 0,Y 62.974,Z 594.818,A -85,B 0,C 180,E1 -28362.912,E2 -28362.912} C_VEL
LIN {X 0,Y 61.686,Z 597.529,A -85,B 0,C 180,E1 -28377.128,E2 -28377.128} C_VEL
LIN {X 0,Y 62.611,Z 598.785,A -85,B 0,C 180,E1 -28388.205,E2 -28388.205} C_VEL
LIN {X 0,Y 65.637,Z 599.447,A -85,B 0,C 180,E1 -28400.021,E2 -28400.021} C_VEL
LIN {X 0,Y 71.647,Z 599.153,A -85,B 0,C 180,E1 -28412.01,E2 -28412.01} C_VEL
LIN {X 0,Y 80.931,Z 597.653,A -85,B 0,C 180,E1 -28422.824,E2 -28422.824} C_VEL
LIN {X 0,Y 92.434,Z 594.812,A -85,B 0,C 180,E1 -28431.326,E2 -28431.326} C_VEL
LIN {X 0,Y 105.507,Z 590.555,A -85,B 0,C 180,E1 -28437.846,E2 -28437.846} C_VEL
LIN {X 0,Y 119.647,Z 584.842,A -85,B 0,C 180,E1 -28442.956,E2 -28442.956} C_VEL
LIN {X 0,Y 134.512,Z 577.56,A -85,B 0,C 180,E1 -28446.881,E2 -28446.881} C_VEL
LIN {X 0,Y 147.93,Z 569.785,A -85,B 0,C 180,E1 -28449.638,E2 -28449.638} C_VEL
LIN {X 0,Y 161.649,Z 560.454,A -85,B 0,C 180,E1 -28451.958,E2 -28451.958} C_VEL
LIN {X 0,Y 165.598,Z 557.41,A -85,B 0,C 180,E1 -28452.53,E2 -28452.53} C_VEL
LIN {X 0,Y 165.909,Z 557.192,A -85,B 0,C 180,E1 -28453.003,E2 -28453.003} C_VEL
LIN {X 0,Y 152.763,Z 566.912,A -85,B 0,C 180,E1 -28454.94,E2 -28454.94} C_VEL
LIN {X 0,Y 138.05,Z 576.197,A -85,B 0,C 180,E1 -28457.568,E2 -28457.568} C_VEL
LIN {X 0,Y 124.1,Z 583.635,A -85,B 0,C 180,E1 -28460.849,E2 -28460.849} C_VEL
LIN {X 0,Y 112,Z 589.174,A -85,B 0,C 180,E1 -28464.496,E2 -28464.496} C_VEL
LIN {X 0,Y 98.86,Z 594.318,A -85,B 0,C 180,E1 -28469.841,E2 -28469.841} C_VEL
LIN {X 0,Y 87.38,Z 597.975,A -85,B 0,C 180,E1 -28476.442,E2 -28476.442} C_VEL
LIN {X 0,Y 78.286,Z 600.412,A -85,B 0,C 180,E1 -28484.08,E2 -28484.08} C_VEL
LIN {X 0,Y 70.834,Z 601.882,A -85,B 0,C 180,E1 -28493.45,E2 -28493.45} C_VEL
LIN {X 0,Y 65.483,Z 602.552,A -85,B 0,C 180,E1 -28504.562,E2 -28504.562} C_VEL
LIN {X 0,Y 62.802,Z 602.247,A -85,B 0,C 180,E1 -28517.051,E2 -28517.051} C_VEL
LIN {X 0,Y 62.45,Z 601.801,A -85,B 0,C 180,E1 -28523.523,E2 -28523.523} C_VEL
LIN {X 0,Y 62.593,Z 601.075,A -85,B 0,C 180,E1 -28529.985,E2 -28529.985} C_VEL
LIN {X 0,Y 62.81,Z 598.75,A -85,B 0,C 180,E1 -28542.915,E2 -28542.915} C_VEL
LIN {X 0,Y 65.459,Z 595.398,A -85,B 0,C 180,E1 -28555.416,E2 -28555.416} C_VEL
LIN {X 0,Y 71.43,Z 590.121,A -85,B 0,C 180,E1 -28568.087,E2 -28568.087} C_VEL
LIN {X 0,Y 79.861,Z 583.41,A -85,B 0,C 180,E1 -28578.398,E2 -28578.398} C_VEL
LIN {X 0,Y 85.232,Z 579.158,A -85,B 0,C 180,E1 -28583.009,E2 -28583.009} C_VEL
LIN {X 0,Y 88.219,Z 576.372,A -85,B 0,C 180,E1 -28585.822,E2 -28585.822} C_VEL
LIN {X 0,Y 96.439,Z 566.255,A -85,B 0,C 180,E1 -28595.105,E2 -28595.105} C_VEL
LIN {X 0,Y 99.906,Z 562.827,A -85,B 0,C 180,E1 -28597.083,E2 -28597.083} C_VEL
LIN {X 0,Y 109.806,Z 553.379,A -85,B 0,C 180,E1 -28600.711,E2 -28600.711} C_VEL
LIN {X 0,Y 120.701,Z 541.745,A -85,B 0,C 180,E1 -28603.854,E2 -28603.854} C_VEL
LIN {X 0,Y 131.129,Z 529.075,A -85,B 0,C 180,E1 -28606.231,E2 -28606.231} C_VEL
LIN {X 0,Y 140.871,Z 515.179,A -85,B 0,C 180,E1 -28608.216,E2 -28608.216} C_VEL
LIN {X 0,Y 149.991,Z 500.014,A -85,B 0,C 180,E1 -28609.682,E2 -28609.682} C_VEL
LIN {X 0,Y 157.48,Z 484.87,A -85,B 0,C 180,E1 -28610.839,E2 -28610.839} C_VEL
LIN {X 0,Y 163.78,Z 469.47,A -85,B 0,C 180,E1 -28611.69,E2 -28611.69} C_VEL
LIN {X 0,Y 168.635,Z 454.8,A -85,B 0,C 180,E1 -28612.29,E2 -28612.29} C_VEL
LIN {X 0,Y 172.785,Z 438.509,A -85,B 0,C 180,E1 -28612.769,E2 -28612.769} C_VEL
LIN {X 0,Y 175.792,Z 420.617,A -85,B 0,C 180,E1 -28613.176,E2 -28613.176} C_VEL
LIN {X 0,Y 180.144,Z 385.078,A -85,B 0,C 180,E1 -28613.908,E2 -28613.908} C_VEL
LIN {X 0,Y 177.484,Z 378.072,A -85,B 0,C 180,E1 -28618.195,E2 -28618.195} C_VEL
LIN {X 0,Y 175.521,Z 372.937,A -85,B 0,C 180,E1 -28622.475,E2 -28622.475} C_VEL
LIN {X 0,Y 174.254,Z 369.592,A -85,B 0,C 180,E1 -28626.464,E2 -28626.464} C_VEL
LIN {X 0,Y 173.488,Z 366.948,A -85,B 0,C 180,E1 -28631.687,E2 -28631.687} C_VEL
LIN {X 0,Y 173.429,Z 367.297,A -85,B 0,C 180,E1 -28635.67,E2 -28635.67} C_VEL
LIN {X 0,Y 174.345,Z 370.532,A -85,B 0,C 180,E1 -28641.705,E2 -28641.705} C_VEL
LIN {X 0,Y 175.878,Z 374.452,A -85,B 0,C 180,E1 -28646.077,E2 -28646.077} C_VEL
LIN {X 0,Y 177.691,Z 378.871,A -85,B 0,C 180,E1 -28649.755,E2 -28649.755} C_VEL
LIN {X 0,Y 180.019,Z 384.972,A -85,B 0,C 180,E1 -28653.467,E2 -28653.467} C_VEL
LIN {X 0,Y 174.788,Z 426.015,A -85,B 0,C 180,E1 -28654.323,E2 -28654.323} C_VEL
LIN {X 0,Y 171.284,Z 442.842,A -85,B 0,C 180,E1 -28654.776,E2 -28654.776} C_VEL
LIN {X 0,Y 166.565,Z 459.326,A -85,B 0,C 180,E1 -28655.439,E2 -28655.439} C_VEL
LIN {X 0,Y 160.774,Z 475.087,A -85,B 0,C 180,E1 -28656.31,E2 -28656.31} C_VEL
LIN {X 0,Y 153.758,Z 490.566,A -85,B 0,C 180,E1 -28657.436,E2 -28657.436} C_VEL
LIN {X 0,Y 145.649,Z 505.425,A -85,B 0,C 180,E1 -28658.852,E2 -28658.852} C_VEL
LIN {X 0,Y 136.533,Z 519.499,A -85,B 0,C 180,E1 -28660.615,E2 -28660.615} C_VEL
LIN {X 0,Y 126.893,Z 532.253,A -85,B 0,C 180,E1 -28662.803,E2 -28662.803} C_VEL
LIN {X 0,Y 117.379,Z 543.251,A -85,B 0,C 180,E1 -28665.304,E2 -28665.304} C_VEL
LIN {X 0,Y 106.673,Z 554.262,A -85,B 0,C 180,E1 -28668.803,E2 -28668.803} C_VEL
LIN {X 0,Y 94.94,Z 564.88,A -85,B 0,C 180,E1 -28673.701,E2 -28673.701} C_VEL
LIN {X 0,Y 83.915,Z 573.759,A -85,B 0,C 180,E1 -28679.848,E2 -28679.848} C_VEL
LIN {X 0,Y 74.018,Z 581.065,A -85,B 0,C 180,E1 -28687.694,E2 -28687.694} C_VEL
LIN {X 0,Y 65.66,Z 587.059,A -85,B 0,C 180,E1 -28697.655,E2 -28697.655} C_VEL
LIN {X 0,Y 59.33,Z 591.881,A -85,B 0,C 180,E1 -28710.016,E2 -28710.016} C_VEL
LIN {X 0,Y 55.471,Z 595.494,A -85,B 0,C 180,E1 -28724.696,E2 -28724.696} C_VEL
LIN {X 0,Y 54.621,Z 597.367,A -85,B 0,C 180,E1 -28735.742,E2 -28735.742} C_VEL
LIN {X 0,Y 55.914,Z 599.004,A -85,B 0,C 180,E1 -28751.042,E2 -28751.042} C_VEL
LIN {X 0,Y 60.068,Z 599.702,A -85,B 0,C 180,E1 -28765.01,E2 -28765.01} C_VEL
LIN {X 0,Y 68.065,Z 599.24,A -85,B 0,C 180,E1 -28778.357,E2 -28778.357} C_VEL
LIN {X 0,Y 80.267,Z 597.235,A -85,B 0,C 180,E1 -28789.912,E2 -28789.912} C_VEL
LIN {X 0,Y 91.53,Z 594.523,A -85,B 0,C 180,E1 -28796.692,E2 -28796.692} C_VEL
LIN {X 0,Y 105.537,Z 590.129,A -85,B 0,C 180,E1 -28802.544,E2 -28802.544} C_VEL
LIN {X 0,Y 120.393,Z 584.222,A -85,B 0,C 180,E1 -28807.03,E2 -28807.03} C_VEL
LIN {X 0,Y 132.669,Z 578.377,A -85,B 0,C 180,E1 -28809.835,E2 -28809.835} C_VEL
LIN {X 0,Y 146.659,Z 570.582,A -85,B 0,C 180,E1 -28812.376,E2 -28812.376} C_VEL
LIN {X 0,Y 144.468,Z 571.946,A -85,B 0,C 180,E1 -28813.338,E2 -28813.338} C_VEL
LIN {X 0,Y 131.352,Z 579.368,A -85,B 0,C 180,E1 -28815.596,E2 -28815.596} C_VEL
LIN {X 0,Y 118.568,Z 585.56,A -85,B 0,C 180,E1 -28818.47,E2 -28818.47} C_VEL
LIN {X 0,Y 103.166,Z 591.841,A -85,B 0,C 180,E1 -28823.104,E2 -28823.104} C_VEL
LIN {X 0,Y 88.707,Z 596.607,A -85,B 0,C 180,E1 -28829.349,E2 -28829.349} C_VEL
LIN {X 0,Y 78.195,Z 599.31,A -85,B 0,C 180,E1 -28835.994,E2 -28835.994} C_VEL
LIN {X 0,Y 66.879,Z 601.531,A -85,B 0,C 180,E1 -28847.353,E2 -28847.353} C_VEL
LIN {X 0,Y 59.098,Z 602.336,A -85,B 0,C 180,E1 -28861.579,E2 -28861.579} C_VEL
LIN {X 0,Y 55.872,Z 601.951,A -85,B 0,C 180,E1 -28875.412,E2 -28875.412} C_VEL
LIN {X 0,Y 55.489,Z 600.716,A -85,B 0,C 180,E1 -28889.983,E2 -28889.983} C_VEL
LIN {X 0,Y 55.861,Z 598.27,A -85,B 0,C 180,E1 -28904.555,E2 -28904.555} C_VEL
LIN {X 0,Y 59.068,Z 594.817,A -85,B 0,C 180,E1 -28918.4,E2 -28918.4} C_VEL
LIN {X 0,Y 65.338,Z 589.825,A -85,B 0,C 180,E1 -28931.158,E2 -28931.158} C_VEL
LIN {X 0,Y 72.965,Z 584.249,A -85,B 0,C 180,E1 -28940.381,E2 -28940.381} C_VEL
LIN {X 0,Y 82.678,Z 577.067,A -85,B 0,C 180,E1 -28948.191,E2 -28948.191} C_VEL
LIN {X 0,Y 93.554,Z 568.325,A -85,B 0,C 180,E1 -28954.323,E2 -28954.323} C_VEL
LIN {X 0,Y 99.906,Z 562.827,A -85,B 0,C 180,E1 -28957.083,E2 -28957.083} C_VEL
LIN {X 0,Y 103.402,Z 559.336,A -85,B 0,C 180,E1 -28958.913,E2 -28958.913} C_VEL
LIN {X 0,Y 108.144,Z 553.39,A -85,B 0,C 180,E1 -28962.368,E2 -28962.368} C_VEL
LIN {X 0,Y 112.963,Z 547.048,A -85,B 0,C 180,E1 -28965.427,E2 -28965.427} C_VEL
LIN {X 0,Y 116.431,Z 542.94,A -85,B 0,C 180,E1 -28966.644,E2 -28966.644} C_VEL
LIN {X 0,Y 127.107,Z 530.478,A -85,B 0,C 180,E1 -28968.89,E2 -28968.89} C_VEL
LIN {X 0,Y 136.893,Z 517.083,A -85,B 0,C 180,E1 -28970.672,E2 -28970.672} C_VEL
LIN {X 0,Y 145.48,Z 503.437,A -85,B 0,C 180,E1 -28971.964,E2 -28971.964} C_VEL
LIN {X 0,Y 153.087,Z 489.132,A -85,B 0,C 180,E1 -28973.034,E2 -28973.034} C_VEL
LIN {X 0,Y 159.895,Z 473.773,A -85,B 0,C 180,E1 -28973.884,E2 -28973.884} C_VEL
LIN {X 0,Y 165.451,Z 458.093,A -85,B 0,C 180,E1 -28974.521,E2 -28974.521} C_VEL
LIN {X 0,Y 169.317,Z 444.227,A -85,B 0,C 180,E1 -28974.905,E2 -28974.905} C_VEL
LIN {X 0,Y 172.697,Z 427.878,A -85,B 0,C 180,E1 -28975.243,E2 -28975.243} C_VEL
LIN {X 0,Y 177.687,Z 389.308,A -85,B 0,C 180,E1 -28975.992,E2 -28975.992} C_VEL
LIN {X 0,Y 175.718,Z 383.849,A -85,B 0,C 180,E1 -28979.558,E2 -28979.558} C_VEL
LIN {X 0,Y 173.998,Z 379.066,A -85,B 0,C 180,E1 -28983.81,E2 -28983.81} C_VEL
LIN {X 0,Y 173.15,Z 376.445,A -85,B 0,C 180,E1 -28986.995,E2 -28986.995} C_VEL
LIN {X 0,Y 172.492,Z 374.001,A -85,B 0,C 180,E1 -28992.118,E2 -28992.118} C_VEL
LIN {X 0,Y 172.454,Z 374.343,A -85,B 0,C 180,E1 -28995.49,E2 -28995.49} C_VEL
LIN {X 0,Y 173.421,Z 378.004,A -85,B 0,C 180,E1 -29001.986,E2 -29001.986} C_VEL
LIN {X 0,Y 174.633,Z 381.276,A -85,B 0,C 180,E1 -29005.551,E2 -29005.551} C_VEL
LIN {X 0,Y 176.263,Z 385.597,A -85,B 0,C 180,E1 -29009.105,E2 -29009.105} C_VEL
LIN {X 0,Y 177.557,Z 389.155,A -85,B 0,C 180,E1 -29011.372,E2 -29011.372} C_VEL
LIN {X 0,Y 172.593,Z 426.973,A -85,B 0,C 180,E1 -29012.101,E2 -29012.101} C_VEL
LIN {X 0,Y 168.881,Z 444.274,A -85,B 0,C 180,E1 -29012.537,E2 -29012.537} C_VEL
LIN {X 0,Y 164.159,Z 460.201,A -85,B 0,C 180,E1 -29013.136,E2 -29013.136} C_VEL
LIN {X 0,Y 158.264,Z 475.82,A -85,B 0,C 180,E1 -29013.931,E2 -29013.931} C_VEL
LIN {X 0,Y 151.127,Z 491.194,A -85,B 0,C 180,E1 -29014.967,E2 -29014.967} C_VEL
LIN {X 0,Y 143.248,Z 505.362,A -85,B 0,C 180,E1 -29016.2,E2 -29016.2} C_VEL
LIN {X 0,Y 133.548,Z 520.018,A -85,B 0,C 180,E1 -29017.887,E2 -29017.887} C_VEL
LIN {X 0,Y 123.678,Z 532.729,A -85,B 0,C 180,E1 -29019.917,E2 -29019.917} C_VEL
LIN {X 0,Y 113.897,Z 543.685,A -85,B 0,C 180,E1 -29022.245,E2 -29022.245} C_VEL
LIN {X 0,Y 102.84,Z 554.656,A -85,B 0,C 180,E1 -29025.55,E2 -29025.55} C_VEL
LIN {X 0,Y 91.527,Z 564.523,A -85,B 0,C 180,E1 -29029.828,E2 -29029.828} C_VEL
LIN {X 0,Y 79.026,Z 574.105,A -85,B 0,C 180,E1 -29036.248,E2 -29036.248} C_VEL
LIN {X 0,Y 69.712,Z 580.536,A -85,B 0,C 180,E1 -29043.038,E2 -29043.038} C_VEL
LIN {X 0,Y 60.418,Z 586.695,A -85,B 0,C 180,E1 -29053.111,E2 -29053.111} C_VEL
LIN {X 0,Y 53.192,Z 591.612,A -85,B 0,C 180,E1 -29066.231,E2 -29066.231} C_VEL
LIN {X 0,Y 49.44,Z 594.544,A -85,B 0,C 180,E1 -29078.192,E2 -29078.192} C_VEL
LIN {X 0,Y 47.528,Z 597.458,A -85,B 0,C 180,E1 -29096.356,E2 -29096.356} C_VEL
LIN {X 0,Y 49.502,Z 599.257,A -85,B 0,C 180,E1 -29115.25,E2 -29115.25} C_VEL
LIN {X 0,Y 55.643,Z 599.919,A -85,B 0,C 180,E1 -29132.178,E2 -29132.178} C_VEL
LIN {X 0,Y 65.373,Z 599.332,A -85,B 0,C 180,E1 -29145.416,E2 -29145.416} C_VEL
LIN {X 0,Y 77.604,Z 597.422,A -85,B 0,C 180,E1 -29155.109,E2 -29155.109} C_VEL
LIN {X 0,Y 91.439,Z 594.206,A -85,B 0,C 180,E1 -29162.1,E2 -29162.1} C_VEL
LIN {X 0,Y 106.272,Z 589.64,A -85,B 0,C 180,E1 -29167.205,E2 -29167.205} C_VEL
LIN {X 0,Y 121.723,Z 583.612,A -85,B 0,C 180,E1 -29170.995,E2 -29170.995} C_VEL
LIN {X 0,Y 129.456,Z 580.068,A -85,B 0,C 180,E1 -29172.54,E2 -29172.54} C_VEL
LIN {X 0,Y 113.279,Z 587.396,A -85,B 0,C 180,E1 -29175.896,E2 -29175.896} C_VEL
LIN {X 0,Y 97.466,Z 593.162,A -85,B 0,C 180,E1 -29180.358,E2 -29180.358} C_VEL
LIN {X 0,Y 85.415,Z 596.714,A -85,B 0,C 180,E1 -29185.143,E2 -29185.143} C_VEL
LIN {X 0,Y 74.192,Z 599.345,A -85,B 0,C 180,E1 -29191.489,E2 -29191.489} C_VEL
LIN {X 0,Y 61.171,Z 601.496,A -85,B 0,C 180,E1 -29203.573,E2 -29203.573} C_VEL
LIN {X 0,Y 52.913,Z 602.096,A -85,B 0,C 180,E1 -29217.888,E2 -29217.888} C_VEL
LIN {X 0,Y 48.976,Z 601.648,A -85,B 0,C 180,E1 -29233.302,E2 -29233.302} C_VEL
LIN {X 0,Y 48.372,Z 600.307,A -85,B 0,C 180,E1 -29249.98,E2 -29249.98} C_VEL
LIN {X 0,Y 48.294,Z 599.201,A -85,B 0,C 180,E1 -29258.347,E2 -29258.347} C_VEL
LIN {X 0,Y 50.466,Z 596.125,A -85,B 0,C 180,E1 -29274.673,E2 -29274.673} C_VEL
LIN {X 0,Y 55.917,Z 592.007,A -85,B 0,C 180,E1 -29288.91,E2 -29288.91} C_VEL
LIN {X 0,Y 66.17,Z 585.088,A -85,B 0,C 180,E1 -29302.778,E2 -29302.778} C_VEL
LIN {X 0,Y 76.361,Z 578.068,A -85,B 0,C 180,E1 -29310.938,E2 -29310.938} C_VEL
LIN {X 0,Y 87.682,Z 569.565,A -85,B 0,C 180,E1 -29317.151,E2 -29317.151} C_VEL
LIN {X 0,Y 99.789,Z 559.388,A -85,B 0,C 180,E1 -29321.912,E2 -29321.912} C_VEL
LIN {X 0,Y 111.253,Z 548.387,A -85,B 0,C 180,E1 -29325.365,E2 -29325.365} C_VEL
LIN {X 0,Y 116.431,Z 542.94,A -85,B 0,C 180,E1 -29326.644,E2 -29326.644} C_VEL
LIN {X 0,Y 119.868,Z 538.804,A -85,B 0,C 180,E1 -29327.77,E2 -29327.77} C_VEL
LIN {X 0,Y 129.316,Z 524.466,A -85,B 0,C 180,E1 -29332.393,E2 -29332.393} C_VEL
LIN {X 0,Y 132.484,Z 519.785,A -85,B 0,C 180,E1 -29333.197,E2 -29333.197} C_VEL
LIN {X 0,Y 141.213,Z 506.708,A -85,B 0,C 180,E1 -29334.393,E2 -29334.393} C_VEL
LIN {X 0,Y 148.936,Z 493.025,A -85,B 0,C 180,E1 -29335.341,E2 -29335.341} C_VEL
LIN {X 0,Y 155.826,Z 478.434,A -85,B 0,C 180,E1 -29336.131,E2 -29336.131} C_VEL
LIN {X 0,Y 161.881,Z 462.792,A -85,B 0,C 180,E1 -29336.749,E2 -29336.749} C_VEL
LIN {X 0,Y 166.878,Z 446.421,A -85,B 0,C 180,E1 -29337.15,E2 -29337.15} C_VEL
LIN {X 0,Y 170.626,Z 429.103,A -85,B 0,C 180,E1 -29337.514,E2 -29337.514} C_VEL
LIN {X 0,Y 175.342,Z 393.494,A -85,B 0,C 180,E1 -29338.171,E2 -29338.171} C_VEL
LIN {X 0,Y 173.897,Z 389.084,A -85,B 0,C 180,E1 -29341.362,E2 -29341.362} C_VEL
LIN {X 0,Y 172.661,Z 385.436,A -85,B 0,C 180,E1 -29344.863,E2 -29344.863} C_VEL
LIN {X 0,Y 172.104,Z 383.396,A -85,B 0,C 180,E1 -29347.325,E2 -29347.325} C_VEL
LIN {X 0,Y 171.537,Z 381.154,A -85,B 0,C 180,E1 -29351.822,E2 -29351.822} C_VEL
LIN {X 0,Y 171.48,Z 381.367,A -85,B 0,C 180,E1 -29355.245,E2 -29355.245} C_VEL
LIN {X 0,Y 172.274,Z 384.76,A -85,B 0,C 180,E1 -29361.363,E2 -29361.363} C_VEL
LIN {X 0,Y 173.415,Z 388.201,A -85,B 0,C 180,E1 -29365.081,E2 -29365.081} C_VEL
LIN {X 0,Y 174.789,Z 392.135,A -85,B 0,C 180,E1 -29368.304,E2 -29368.304} C_VEL
LIN {X 0,Y 175.215,Z 393.445,A -85,B 0,C 180,E1 -29369.175,E2 -29369.175} C_VEL
LIN {X 0,Y 171.34,Z 423.221,A -85,B 0,C 180,E1 -29369.759,E2 -29369.759} C_VEL
LIN {X 0,Y 167.981,Z 440.222,A -85,B 0,C 180,E1 -29370.113,E2 -29370.113} C_VEL
LIN {X 0,Y 163.291,Z 456.968,A -85,B 0,C 180,E1 -29370.609,E2 -29370.609} C_VEL
LIN {X 0,Y 157.74,Z 472.352,A -85,B 0,C 180,E1 -29371.269,E2 -29371.269} C_VEL
LIN {X 0,Y 150.495,Z 488.405,A -85,B 0,C 180,E1 -29372.191,E2 -29372.191} C_VEL
LIN {X 0,Y 141.871,Z 503.985,A -85,B 0,C 180,E1 -29373.364,E2 -29373.364} C_VEL
LIN {X 0,Y 132.571,Z 518.019,A -85,B 0,C 180,E1 -29374.761,E2 -29374.761} C_VEL
LIN {X 0,Y 122.474,Z 531.077,A -85,B 0,C 180,E1 -29376.563,E2 -29376.563} C_VEL
LIN {X 0,Y 111.342,Z 543.434,A -85,B 0,C 180,E1 -29378.87,E2 -29378.87} C_VEL
LIN {X 0,Y 100.964,Z 553.564,A -85,B 0,C 180,E1 -29381.574,E2 -29381.574} C_VEL
LIN {X 0,Y 89.751,Z 563.072,A -85,B 0,C 180,E1 -29385.208,E2 -29385.208} C_VEL
LIN {X 0,Y 77.429,Z 572.292,A -85,B 0,C 180,E1 -29390.57,E2 -29390.57} C_VEL
LIN {X 0,Y 65.922,Z 579.962,A -85,B 0,C 180,E1 -29397.807,E2 -29397.807} C_VEL
LIN {X 0,Y 55.636,Z 586.294,A -85,B 0,C 180,E1 -29407.75,E2 -29407.75} C_VEL
LIN {X 0,Y 47.338,Z 591.294,A -85,B 0,C 180,E1 -29421.483,E2 -29421.483} C_VEL
LIN {X 0,Y 41.815,Z 595.196,A -85,B 0,C 180,E1 -29439.699,E2 -29439.699} C_VEL
LIN {X 0,Y 40.422,Z 597.827,A -85,B 0,C 180,E1 -29459.61,E2 -29459.61} C_VEL
LIN {X 0,Y 43.028,Z 599.423,A -85,B 0,C 180,E1 -29479.199,E2 -29479.199} C_VEL
LIN {X 0,Y 48.547,Z 600.087,A -85,B 0,C 180,E1 -29494.255,E2 -29494.255} C_VEL
LIN {X 0,Y 57.656,Z 599.895,A -85,B 0,C 180,E1 -29507.271,E2 -29507.271} C_VEL
LIN {X 0,Y 70.355,Z 598.523,A -85,B 0,C 180,E1 -29517.613,E2 -29517.613} C_VEL
LIN {X 0,Y 84.681,Z 595.778,A -85,B 0,C 180,E1 -29524.758,E2 -29524.758} C_VEL
LIN {X 0,Y 99.852,Z 591.715,A -85,B 0,C 180,E1 -29529.766,E2 -29529.766} C_VEL
LIN {X 0,Y 109.655,Z 588.465,A -85,B 0,C 180,E1 -29532.21,E2 -29532.21} C_VEL
LIN {X 0,Y 108.227,Z 589.015,A -85,B 0,C 180,E1 -29533.049,E2 -29533.049} C_VEL
LIN {X 0,Y 95.212,Z 593.447,A -85,B 0,C 180,E1 -29536.316,E2 -29536.316} C_VEL
LIN {X 0,Y 82.622,Z 596.833,A -85,B 0,C 180,E1 -29540.635,E2 -29540.635} C_VEL
LIN {X 0,Y 70.698,Z 599.382,A -85,B 0,C 180,E1 -29546.506,E2 -29546.506} C_VEL
LIN {X 0,Y 55.019,Z 601.552,A -85,B 0,C 180,E1 -29559.942,E2 -29559.942} C_VEL
LIN {X 0,Y 44.071,Z 601.729,A -85,B 0,C 180,E1 -29581.394,E2 -29581.394} C_VEL
LIN {X 0,Y 41.29,Z 600.716,A -85,B 0,C 180,E1 -29600.176,E2 -29600.176} C_VEL
LIN {X 0,Y 41.274,Z 599.876,A -85,B 0,C 180,E1 -29609.977,E2 -29609.977} C_VEL
LIN {X 0,Y 41.244,Z 598.748,A -85,B 0,C 180,E1 -29619.787,E2 -29619.787} C_VEL
LIN {X 0,Y 44.048,Z 595.557,A -85,B 0,C 180,E1 -29638.572,E2 -29638.572} C_VEL
LIN {X 0,Y 50.515,Z 591.3,A -85,B 0,C 180,E1 -29654.049,E2 -29654.049} C_VEL
LIN {X 0,Y 59.507,Z 585.812,A -85,B 0,C 180,E1 -29665.732,E2 -29665.732} C_VEL
LIN {X 0,Y 70.241,Z 578.991,A -85,B 0,C 180,E1 -29674.187,E2 -29674.187} C_VEL
LIN {X 0,Y 82.052,Z 570.752,A -85,B 0,C 180,E1 -29680.379,E2 -29680.379} C_VEL
LIN {X 0,Y 92.982,Z 562.23,A -85,B 0,C 180,E1 -29684.467,E2 -29684.467} C_VEL
LIN {X 0,Y 104.262,Z 552.143,A -85,B 0,C 180,E1 -29687.741,E2 -29687.741} C_VEL
LIN {X 0,Y 115.827,Z 540.344,A -85,B 0,C 180,E1 -29690.338,E2 -29690.338} C_VEL
LIN {X 0,Y 126.755,Z 527.467,A -85,B 0,C 180,E1 -29692.27,E2 -29692.27} C_VEL
LIN {X 0,Y 132.484,Z 519.785,A -85,B 0,C 180,E1 -29693.197,E2 -29693.197} C_VEL
LIN {X 0,Y 135.581,Z 515.102,A -85,B 0,C 180,E1 -29693.944,E2 -29693.944} C_VEL
LIN {X 0,Y 143.004,Z 500.807,A -85,B 0,C 180,E1 -29697.102,E2 -29697.102} C_VEL
LIN {X 0,Y 145.579,Z 495.727,A -85,B 0,C 180,E1 -29697.796,E2 -29697.796} C_VEL
LIN {X 0,Y 146.499,Z 493.976,A -85,B 0,C 180,E1 -29697.925,E2 -29697.925} C_VEL
LIN {X 0,Y 153.758,Z 479.013,A -85,B 0,C 180,E1 -29698.643,E2 -29698.643} C_VEL
LIN {X 0,Y 159.881,Z 463.619,A -85,B 0,C 180,E1 -29699.162,E2 -29699.162} C_VEL
LIN {X 0,Y 165.14,Z 446.722,A -85,B 0,C 180,E1 -29699.52,E2 -29699.52} C_VEL
LIN {X 0,Y 168.87,Z 429.854,A -85,B 0,C 180,E1 -29699.833,E2 -29699.833} C_VEL
LIN {X 0,Y 173.237,Z 397.918,A -85,B 0,C 180,E1 -29700.385,E2 -29700.385} C_VEL
LIN {X 0,Y 171.742,Z 392.923,A -85,B 0,C 180,E1 -29704.591,E2 -29704.591} C_VEL
LIN {X 0,Y 171.06,Z 390.313,A -85,B 0,C 180,E1 -29707.694,E2 -29707.694} C_VEL
LIN {X 0,Y 170.566,Z 388.225,A -85,B 0,C 180,E1 -29711.89,E2 -29711.89} C_VEL
LIN {X 0,Y 170.507,Z 388.41,A -85,B 0,C 180,E1 -29714.997,E2 -29714.997} C_VEL
LIN {X 0,Y 171.17,Z 391.636,A -85,B 0,C 180,E1 -29720.861,E2 -29720.861} C_VEL
LIN {X 0,Y 172.177,Z 394.976,A -85,B 0,C 180,E1 -29724.501,E2 -29724.501} C_VEL
LIN {X 0,Y 173.157,Z 397.933,A -85,B 0,C 180,E1 -29727.007,E2 -29727.007} C_VEL
LIN {X 0,Y 169.083,Z 427.567,A -85,B 0,C 180,E1 -29727.502,E2 -29727.502} C_VEL
LIN {X 0,Y 165.272,Z 444.837,A -85,B 0,C 180,E1 -29727.84,E2 -29727.84} C_VEL
LIN {X 0,Y 160.223,Z 461.319,A -85,B 0,C 180,E1 -29728.34,E2 -29728.34} C_VEL
LIN {X 0,Y 154.106,Z 476.884,A -85,B 0,C 180,E1 -29728.967,E2 -29728.967} C_VEL
LIN {X 0,Y 146.751,Z 492.124,A -85,B 0,C 180,E1 -29729.788,E2 -29729.788} C_VEL
LIN {X 0,Y 138.119,Z 506.943,A -85,B 0,C 180,E1 -29730.813,E2 -29730.813} C_VEL
LIN {X 0,Y 128.547,Z 520.795,A -85,B 0,C 180,E1 -29732.085,E2 -29732.085} C_VEL
LIN {X 0,Y 118.253,Z 533.47,A -85,B 0,C 180,E1 -29733.709,E2 -29733.709} C_VEL
LIN {X 0,Y 107.526,Z 544.854,A -85,B 0,C 180,E1 -29735.706,E2 -29735.706} C_VEL
LIN {X 0,Y 96.276,Z 555.292,A -85,B 0,C 180,E1 -29738.323,E2 -29738.323} C_VEL
LIN {X 0,Y 84.219,Z 565.037,A -85,B 0,C 180,E1 -29741.885,E2 -29741.885} C_VEL
LIN {X 0,Y 70.352,Z 574.684,A -85,B 0,C 180,E1 -29747.62,E2 -29747.62} C_VEL
LIN {X 0,Y 56.939,Z 582.787,A -85,B 0,C 180,E1 -29756.281,E2 -29756.281} C_VEL
LIN {X 0,Y 44.833,Z 589.423,A -85,B 0,C 180,E1 -29770.158,E2 -29770.158} C_VEL
LIN {X 0,Y 39.865,Z 592.133,A -85,B 0,C 180,E1 -29779.871,E2 -29779.871} C_VEL
LIN {X 0,Y 34.181,Z 595.85,A -85,B 0,C 180,E1 -29801.894,E2 -29801.894} C_VEL
LIN {X 0,Y 33.413,Z 598.041,A -85,B 0,C 180,E1 -29822.705,E2 -29822.705} C_VEL
LIN {X 0,Y 37.03,Z 599.621,A -85,B 0,C 180,E1 -29845.286,E2 -29845.286} C_VEL
LIN {X 0,Y 44.321,Z 600.323,A -85,B 0,C 180,E1 -29862.132,E2 -29862.132} C_VEL
LIN {X 0,Y 56.389,Z 599.993,A -85,B 0,C 180,E1 -29875.813,E2 -29875.813} C_VEL
LIN {X 0,Y 70.526,Z 598.438,A -85,B 0,C 180,E1 -29884.645,E2 -29884.645} C_VEL
LIN {X 0,Y 85.78,Z 595.6,A -85,B 0,C 180,E1 -29890.478,E2 -29890.478} C_VEL
LIN {X 0,Y 91.644,Z 594.142,A -85,B 0,C 180,E1 -29892.16,E2 -29892.16} C_VEL
LIN {X 0,Y 86.863,Z 595.449,A -85,B 0,C 180,E1 -29893.816,E2 -29893.816} C_VEL
LIN {X 0,Y 67.792,Z 599.419,A -85,B 0,C 180,E1 -29901.053,E2 -29901.053} C_VEL
LIN {X 0,Y 50.712,Z 601.39,A -85,B 0,C 180,E1 -29913.715,E2 -29913.715} C_VEL
LIN {X 0,Y 41.458,Z 601.612,A -85,B 0,C 180,E1 -29927.276,E2 -29927.276} C_VEL
LIN {X 0,Y 35.511,Z 601.033,A -85,B 0,C 180,E1 -29946.654,E2 -29946.654} C_VEL
LIN {X 0,Y 34.281,Z 600.348,A -85,B 0,C 180,E1 -29958.141,E2 -29958.141} C_VEL
LIN {X 0,Y 34.154,Z 599.443,A -85,B 0,C 180,E1 -29969.972,E2 -29969.972} C_VEL
LIN {X 0,Y 35.477,Z 596.786,A -85,B 0,C 180,E1 -29993.31,E2 -29993.31} C_VEL
LIN {X 0,Y 41.392,Z 592.927,A -85,B 0,C 180,E1 -30012.744,E2 -30012.744} C_VEL
LIN {X 0,Y 50.432,Z 587.949,A -85,B 0,C 180,E1 -30026.696,E2 -30026.696} C_VEL
LIN {X 0,Y 61.436,Z 581.695,A -85,B 0,C 180,E1 -30036.184,E2 -30036.184} C_VEL
LIN {X 0,Y 75.495,Z 572.738,A -85,B 0,C 180,E1 -30043.601,E2 -30043.601} C_VEL
LIN {X 0,Y 88.023,Z 563.549,A -85,B 0,C 180,E1 -30047.915,E2 -30047.915} C_VEL
LIN {X 0,Y 99.607,Z 553.768,A -85,B 0,C 180,E1 -30050.966,E2 -30050.966} C_VEL
LIN {X 0,Y 109.722,Z 544.102,A -85,B 0,C 180,E1 -30053.022,E2 -30053.022} C_VEL
LIN {X 0,Y 119.97,Z 532.868,A -85,B 0,C 180,E1 -30054.687,E2 -30054.687} C_VEL
LIN {X 0,Y 130.291,Z 519.774,A -85,B 0,C 180,E1 -30056.142,E2 -30056.142} C_VEL
LIN {X 0,Y 139.515,Z 506.144,A -85,B 0,C 180,E1 -30057.196,E2 -30057.196} C_VEL
LIN {X 0,Y 146.499,Z 493.976,A -85,B 0,C 180,E1 -30057.925,E2 -30057.925} C_VEL
LIN {X 0,Y 149.041,Z 488.828,A -85,B 0,C 180,E1 -30058.432,E2 -30058.432} C_VEL
LIN {X 0,Y 154.983,Z 473.316,A -85,B 0,C 180,E1 -30060.905,E2 -30060.905} C_VEL
LIN {X 0,Y 156.845,Z 467.93,A -85,B 0,C 180,E1 -30061.487,E2 -30061.487} C_VEL
LIN {X 0,Y 157.526,Z 466.101,A -85,B 0,C 180,E1 -30061.582,E2 -30061.582} C_VEL
LIN {X 0,Y 162.728,Z 450.202,A -85,B 0,C 180,E1 -30061.889,E2 -30061.889} C_VEL
LIN {X 0,Y 166.838,Z 433.193,A -85,B 0,C 180,E1 -30062.152,E2 -30062.152} C_VEL
LIN {X 0,Y 169.936,Z 413.323,A -85,B 0,C 180,E1 -30062.457,E2 -30062.457} C_VEL
LIN {X 0,Y 171.33,Z 402.526,A -85,B 0,C 180,E1 -30062.65,E2 -30062.65} C_VEL
LIN {X 0,Y 170.345,Z 398.949,A -85,B 0,C 180,E1 -30066.097,E2 -30066.097} C_VEL
LIN {X 0,Y 169.937,Z 397.117,A -85,B 0,C 180,E1 -30068.395,E2 -30068.395} C_VEL
LIN {X 0,Y 169.595,Z 395.303,A -85,B 0,C 180,E1 -30071.96,E2 -30071.96} C_VEL
LIN {X 0,Y 169.539,Z 395.437,A -85,B 0,C 180,E1 -30074.744,E2 -30074.744} C_VEL
LIN {X 0,Y 170.101,Z 398.585,A -85,B 0,C 180,E1 -30080.466,E2 -30080.466} C_VEL
LIN {X 0,Y 170.946,Z 401.769,A -85,B 0,C 180,E1 -30083.897,E2 -30083.897} C_VEL
LIN {X 0,Y 171.223,Z 402.617,A -85,B 0,C 180,E1 -30084.705,E2 -30084.705} C_VEL
LIN {X 0,Y 170.252,Z 410.331,A -85,B 0,C 180,E1 -30084.894,E2 -30084.894} C_VEL
LIN {X 0,Y 167.01,Z 431.264,A -85,B 0,C 180,E1 -30085.187,E2 -30085.187} C_VEL
LIN {X 0,Y 162.988,Z 448.094,A -85,B 0,C 180,E1 -30085.487,E2 -30085.487} C_VEL
LIN {X 0,Y 157.735,Z 464.383,A -85,B 0,C 180,E1 -30085.93,E2 -30085.93} C_VEL
LIN {X 0,Y 151.162,Z 480.307,A -85,B 0,C 180,E1 -30086.511,E2 -30086.511} C_VEL
LIN {X 0,Y 143.263,Z 495.741,A -85,B 0,C 180,E1 -30087.252,E2 -30087.252} C_VEL
LIN {X 0,Y 134.763,Z 509.581,A -85,B 0,C 180,E1 -30088.11,E2 -30088.11} C_VEL
LIN {X 0,Y 124.81,Z 523.329,A -85,B 0,C 180,E1 -30089.235,E2 -30089.235} C_VEL
LIN {X 0,Y 114.373,Z 535.705,A -85,B 0,C 180,E1 -30090.673,E2 -30090.673} C_VEL
LIN {X 0,Y 102.216,Z 548.008,A -85,B 0,C 180,E1 -30092.64,E2 -30092.64} C_VEL
LIN {X 0,Y 90.209,Z 558.39,A -85,B 0,C 180,E1 -30095.134,E2 -30095.134} C_VEL
LIN {X 0,Y 78.329,Z 567.287,A -85,B 0,C 180,E1 -30098.294,E2 -30098.294} C_VEL
LIN {X 0,Y 66.72,Z 574.942,A -85,B 0,C 180,E1 -30102.518,E2 -30102.518} C_VEL
LIN {X 0,Y 54.002,Z 582.185,A -85,B 0,C 180,E1 -30109.43,E2 -30109.43} C_VEL
LIN {X 0,Y 42.237,Z 588.118,A -85,B 0,C 180,E1 -30120.082,E2 -30120.082} C_VEL
LIN {X 0,Y 34.64,Z 591.786,A -85,B 0,C 180,E1 -30132.312,E2 -30132.312} C_VEL
LIN {X 0,Y 28.161,Z 595.225,A -85,B 0,C 180,E1 -30153.253,E2 -30153.253} C_VEL
LIN {X 0,Y 26.538,Z 598.242,A -85,B 0,C 180,E1 -30187.38,E2 -30187.38} C_VEL
LIN {X 0,Y 31.605,Z 599.82,A -85,B 0,C 180,E1 -30213.586,E2 -30213.586} C_VEL
LIN {X 0,Y 42.489,Z 600.603,A -85,B 0,C 180,E1 -30233.125,E2 -30233.125} C_VEL
LIN {X 0,Y 56.421,Z 600.1,A -85,B 0,C 180,E1 -30244.61,E2 -30244.61} C_VEL
LIN {X 0,Y 71.748,Z 598.352,A -85,B 0,C 180,E1 -30251.554,E2 -30251.554} C_VEL
LIN {X 0,Y 72.088,Z 598.339,A -85,B 0,C 180,E1 -30252.809,E2 -30252.809} C_VEL
LIN {X 0,Y 59.182,Z 600.239,A -85,B 0,C 180,E1 -30258.147,E2 -30258.147} C_VEL
LIN {X 0,Y 41.545,Z 601.439,A -85,B 0,C 180,E1 -30272.2,E2 -30272.2} C_VEL
LIN {X 0,Y 29.067,Z 600.661,A -85,B 0,C 180,E1 -30301.044,E2 -30301.044} C_VEL
LIN {X 0,Y 27.325,Z 599.968,A -85,B 0,C 180,E1 -30315.06,E2 -30315.06} C_VEL
LIN {X 0,Y 27.034,Z 598.999,A -85,B 0,C 180,E1 -30329.964,E2 -30329.964} C_VEL
LIN {X 0,Y 29.029,Z 596.215,A -85,B 0,C 180,E1 -30358.921,E2 -30358.921} C_VEL
LIN {X 0,Y 36.437,Z 592.272,A -85,B 0,C 180,E1 -30380.445,E2 -30380.445} C_VEL
LIN {X 0,Y 46.865,Z 587.145,A -85,B 0,C 180,E1 -30394.077,E2 -30394.077} C_VEL
LIN {X 0,Y 58.883,Z 580.793,A -85,B 0,C 180,E1 -30402.653,E2 -30402.653} C_VEL
LIN {X 0,Y 71.746,Z 572.959,A -85,B 0,C 180,E1 -30408.319,E2 -30408.319} C_VEL
LIN {X 0,Y 85.105,Z 563.573,A -85,B 0,C 180,E1 -30412.193,E2 -30412.193} C_VEL
LIN {X 0,Y 97.011,Z 553.834,A -85,B 0,C 180,E1 -30414.819,E2 -30414.819} C_VEL
LIN {X 0,Y 109.084,Z 542.458,A -85,B 0,C 180,E1 -30416.792,E2 -30416.792} C_VEL
LIN {X 0,Y 120.389,Z 530.028,A -85,B 0,C 180,E1 -30418.242,E2 -30418.242} C_VEL
LIN {X 0,Y 130.881,Z 516.398,A -85,B 0,C 180,E1 -30419.419,E2 -30419.419} C_VEL
LIN {X 0,Y 139.357,Z 503.544,A -85,B 0,C 180,E1 -30420.166,E2 -30420.166} C_VEL
LIN {X 0,Y 147.582,Z 488.775,A -85,B 0,C 180,E1 -30420.873,E2 -30420.873} C_VEL
LIN {X 0,Y 154.639,Z 473.476,A -85,B 0,C 180,E1 -30421.399,E2 -30421.399} C_VEL
LIN {X 0,Y 157.526,Z 466.101,A -85,B 0,C 180,E1 -30421.582,E2 -30421.582} C_VEL
LIN {X 0,Y 159.43,Z 460.591,A -85,B 0,C 180,E1 -30421.988,E2 -30421.988} C_VEL
LIN {X 0,Y 161.831,Z 451.541,A -85,B 0,C 180,E1 -30423.207,E2 -30423.207} C_VEL
LIN {X 0,Y 163.817,Z 442.336,A -85,B 0,C 180,E1 -30424.301,E2 -30424.301} C_VEL
LIN {X 0,Y 165.005,Z 436.592,A -85,B 0,C 180,E1 -30424.524,E2 -30424.524} C_VEL
LIN {X 0,Y 167.942,Z 420.035,A -85,B 0,C 180,E1 -30424.736,E2 -30424.736} C_VEL
LIN {X 0,Y 169.607,Z 407.432,A -85,B 0,C 180,E1 -30424.931,E2 -30424.931} C_VEL
LIN {X 0,Y 168.902,Z 404.07,A -85,B 0,C 180,E1 -30428.73,E2 -30428.73} C_VEL
LIN {X 0,Y 168.617,Z 402.43,A -85,B 0,C 180,E1 -30432.03,E2 -30432.03} C_VEL
LIN {X 0,Y 168.554,Z 402.692,A -85,B 0,C 180,E1 -30434.917,E2 -30434.917} C_VEL
LIN {X 0,Y 169.016,Z 405.428,A -85,B 0,C 180,E1 -30439.944,E2 -30439.944} C_VEL
LIN {X 0,Y 169.523,Z 407.608,A -85,B 0,C 180,E1 -30442.442,E2 -30442.442} C_VEL
LIN {X 0,Y 166.459,Z 428.57,A -85,B 0,C 180,E1 -30442.737,E2 -30442.737} C_VEL
LIN {X 0,Y 162.597,Z 445.641,A -85,B 0,C 180,E1 -30442.978,E2 -30442.978} C_VEL
LIN {X 0,Y 157.358,Z 462.281,A -85,B 0,C 180,E1 -30443.332,E2 -30443.332} C_VEL
LIN {X 0,Y 150.709,Z 478.629,A -85,B 0,C 180,E1 -30443.791,E2 -30443.791} C_VEL
LIN {X 0,Y 142.736,Z 494.42,A -85,B 0,C 180,E1 -30444.391,E2 -30444.391} C_VEL
LIN {X 0,Y 133.853,Z 508.966,A -85,B 0,C 180,E1 -30445.102,E2 -30445.102} C_VEL
LIN {X 0,Y 124.065,Z 522.491,A -85,B 0,C 180,E1 -30445.959,E2 -30445.959} C_VEL
LIN {X 0,Y 114.348,Z 534.038,A -85,B 0,C 180,E1 -30446.999,E2 -30446.999} C_VEL
LIN {X 0,Y 103.732,Z 544.902,A -85,B 0,C 180,E1 -30448.289,E2 -30448.289} C_VEL
LIN {X 0,Y 91.446,Z 555.813,A -85,B 0,C 180,E1 -30450.187,E2 -30450.187} C_VEL
LIN {X 0,Y 80.093,Z 564.519,A -85,B 0,C 180,E1 -30452.367,E2 -30452.367} C_VEL
LIN {X 0,Y 67.097,Z 573.078,A -85,B 0,C 180,E1 -30455.759,E2 -30455.759} C_VEL
LIN {X 0,Y 53.498,Z 580.746,A -85,B 0,C 180,E1 -30461.065,E2 -30461.065} C_VEL
LIN {X 0,Y 42.14,Z 586.293,A -85,B 0,C 180,E1 -30468.188,E2 -30468.188} C_VEL
LIN {X 0,Y 30.194,Z 591.438,A -85,B 0,C 180,E1 -30482.293,E2 -30482.293} C_VEL
LIN {X 0,Y 21.046,Z 595.495,A -85,B 0,C 180,E1 -30510.046,E2 -30510.046} C_VEL
LIN {X 0,Y 19.081,Z 597.122,A -85,B 0,C 180,E1 -30531.666,E2 -30531.666} C_VEL
LIN {X 0,Y 19.949,Z 598.437,A -85,B 0,C 180,E1 -30555.188,E2 -30555.188} C_VEL
LIN {X 0,Y 28.716,Z 600.186,A -85,B 0,C 180,E1 -30588.381,E2 -30588.381} C_VEL
LIN {X 0,Y 42.324,Z 600.804,A -85,B 0,C 180,E1 -30604.673,E2 -30604.673} C_VEL
LIN {X 0,Y 53.264,Z 600.468,A -85,B 0,C 180,E1 -30611.248,E2 -30611.248} C_VEL
LIN {X 0,Y 50.775,Z 600.72,A -85,B 0,C 180,E1 -30614.258,E2 -30614.258} C_VEL
LIN {X 0,Y 38.21,Z 601.197,A -85,B 0,C 180,E1 -30623.064,E2 -30623.064} C_VEL
LIN {X 0,Y 27.208,Z 600.792,A -85,B 0,C 180,E1 -30639.149,E2 -30639.149} C_VEL
LIN {X 0,Y 20.513,Z 599.573,A -85,B 0,C 180,E1 -30669.915,E2 -30669.915} C_VEL
LIN {X 0,Y 19.93,Z 598.552,A -85,B 0,C 180,E1 -30689.951,E2 -30689.951} C_VEL
LIN {X 0,Y 23.023,Z 595.619,A -85,B 0,C 180,E1 -30727.572,E2 -30727.572} C_VEL
LIN {X 0,Y 32.327,Z 591.598,A -85,B 0,C 180,E1 -30750.348,E2 -30750.348} C_VEL
LIN {X 0,Y 44.189,Z 586.313,A -85,B 0,C 180,E1 -30762.525,E2 -30762.525} C_VEL
LIN {X 0,Y 57.143,Z 579.79,A -85,B 0,C 180,E1 -30769.603,E2 -30769.603} C_VEL
LIN {X 0,Y 70.638,Z 571.866,A -85,B 0,C 180,E1 -30774.071,E2 -30774.071} C_VEL
LIN {X 0,Y 84.425,Z 562.278,A -85,B 0,C 180,E1 -30777.085,E2 -30777.085} C_VEL
LIN {X 0,Y 96.626,Z 552.32,A -85,B 0,C 180,E1 -30779.104,E2 -30779.104} C_VEL
LIN {X 0,Y 108.919,Z 540.677,A -85,B 0,C 180,E1 -30780.618,E2 -30780.618} C_VEL
LIN {X 0,Y 120.385,Z 527.987,A -85,B 0,C 180,E1 -30781.693,E2 -30781.693} C_VEL
LIN {X 0,Y 131.01,Z 514.076,A -85,B 0,C 180,E1 -30782.606,E2 -30782.606} C_VEL
LIN {X 0,Y 140.759,Z 498.891,A -85,B 0,C 180,E1 -30783.213,E2 -30783.213} C_VEL
LIN {X 0,Y 148.759,Z 483.719,A -85,B 0,C 180,E1 -30783.729,E2 -30783.729} C_VEL
LIN {X 0,Y 155.426,Z 468.282,A -85,B 0,C 180,E1 -30784.08,E2 -30784.08} C_VEL
LIN {X 0,Y 160.763,Z 452.798,A -85,B 0,C 180,E1 -30784.334,E2 -30784.334} C_VEL
LIN {X 0,Y 165.005,Z 436.592,A -85,B 0,C 180,E1 -30784.524,E2 -30784.524} C_VEL
LIN {X 0,Y 165.708,Z 432.746,A -85,B 0,C 180,E1 -30784.76,E2 -30784.76} C_VEL
LIN {X 0,Y 166.456,Z 426.775,A -85,B 0,C 180,E1 -30785.815,E2 -30785.815} C_VEL
LIN {X 0,Y 167.084,Z 420.785,A -85,B 0,C 180,E1 -30786.898,E2 -30786.898} C_VEL
LIN {X 0,Y 167.555,Z 416.894,A -85,B 0,C 180,E1 -30787.175,E2 -30787.175} C_VEL
LIN {X 0,Y 168.124,Z 412.525,A -85,B 0,C 180,E1 -30787.285,E2 -30787.285} C_VEL
LIN {X 0,Y 167.794,Z 410.726,A -85,B 0,C 180,E1 -30789.646,E2 -30789.646} C_VEL
LIN {X 0,Y 167.643,Z 409.531,A -85,B 0,C 180,E1 -30792.101,E2 -30792.101} C_VEL
LIN {X 0,Y 167.58,Z 409.801,A -85,B 0,C 180,E1 -30794.79,E2 -30794.79} C_VEL
LIN {X 0,Y 167.975,Z 412.534,A -85,B 0,C 180,E1 -30799.716,E2 -30799.716} C_VEL
LIN {X 0,Y 168.052,Z 412.857,A -85,B 0,C 180,E1 -30800.129,E2 -30800.129} C_VEL
LIN {X 0,Y 165.038,Z 431.682,A -85,B 0,C 180,E1 -30800.337,E2 -30800.337} C_VEL
LIN {X 0,Y 160.923,Z 448.626,A -85,B 0,C 180,E1 -30800.534,E2 -30800.534} C_VEL
LIN {X 0,Y 155.52,Z 465.032,A -85,B 0,C 180,E1 -30800.816,E2 -30800.816} C_VEL
LIN {X 0,Y 148.826,Z 480.929,A -85,B 0,C 180,E1 -30801.171,E2 -30801.171} C_VEL
LIN {X 0,Y 140.785,Z 496.319,A -85,B 0,C 180,E1 -30801.626,E2 -30801.626} C_VEL
LIN {X 0,Y 131.862,Z 510.504,A -85,B 0,C 180,E1 -30802.144,E2 -30802.144} C_VEL
LIN {X 0,Y 121.947,Z 523.852,A -85,B 0,C 180,E1 -30802.79,E2 -30802.79} C_VEL
LIN {X 0,Y 111.226,Z 536.211,A -85,B 0,C 180,E1 -30803.649,E2 -30803.649} C_VEL
LIN {X 0,Y 98.695,Z 548.499,A -85,B 0,C 180,E1 -30804.809,E2 -30804.809} C_VEL
LIN {X 0,Y 86.197,Z 558.878,A -85,B 0,C 180,E1 -30806.28,E2 -30806.28} C_VEL
LIN {X 0,Y 74.985,Z 566.927,A -85,B 0,C 180,E1 -30807.949,E2 -30807.949} C_VEL
LIN {X 0,Y 61.318,Z 575.399,A -85,B 0,C 180,E1 -30810.761,E2 -30810.761} C_VEL
LIN {X 0,Y 47.632,Z 582.469,A -85,B 0,C 180,E1 -30815.064,E2 -30815.064} C_VEL
LIN {X 0,Y 33.568,Z 588.558,A -85,B 0,C 180,E1 -30822.925,E2 -30822.925} C_VEL
LIN {X 0,Y 23.734,Z 592.232,A -85,B 0,C 180,E1 -30833.736,E2 -30833.736} C_VEL
LIN {X 0,Y 13.225,Z 596.116,A -85,B 0,C 180,E1 -30870.073,E2 -30870.073} C_VEL
LIN {X 0,Y 14.036,Z 598.612,A -85,B 0,C 180,E1 -30929.937,E2 -30929.937} C_VEL
LIN {X 0,Y 24.022,Z 600.202,A -85,B 0,C 180,E1 -30959.991,E2 -30959.991} C_VEL
LIN {X 0,Y 35.901,Z 600.935,A -85,B 0,C 180,E1 -30971.693,E2 -30971.693} C_VEL
LIN {X 0,Y 36.004,Z 600.952,A -85,B 0,C 180,E1 -30972.46,E2 -30972.46} C_VEL
LIN {X 0,Y 23.354,Z 600.474,A -85,B 0,C 180,E1 -30985.381,E2 -30985.381} C_VEL
LIN {X 0,Y 14.036,Z 599.114,A -85,B 0,C 180,E1 -31019.874,E2 -31019.874} C_VEL
LIN {X 0,Y 12.811,Z 598.098,A -85,B 0,C 180,E1 -31049.924,E2 -31049.924} C_VEL
LIN {X 0,Y 17.894,Z 595.021,A -85,B 0,C 180,E1 -31101.678,E2 -31101.678} C_VEL
LIN {X 0,Y 29.431,Z 590.893,A -85,B 0,C 180,E1 -31122.665,E2 -31122.665} C_VEL
LIN {X 0,Y 42.577,Z 585.478,A -85,B 0,C 180,E1 -31131.871,E2 -31131.871} C_VEL
LIN {X 0,Y 56.289,Z 578.787,A -85,B 0,C 180,E1 -31136.868,E2 -31136.868} C_VEL
LIN {X 0,Y 70.615,Z 570.464,A -85,B 0,C 180,E1 -31140.003,E2 -31140.003} C_VEL
LIN {X 0,Y 84.366,Z 560.98,A -85,B 0,C 180,E1 -31141.987,E2 -31141.987} C_VEL
LIN {X 0,Y 96.785,Z 550.803,A -85,B 0,C 180,E1 -31143.407,E2 -31143.407} C_VEL
LIN {X 0,Y 109.238,Z 538.906,A -85,B 0,C 180,E1 -31144.42,E2 -31144.42} C_VEL
LIN {X 0,Y 120.815,Z 525.912,A -85,B 0,C 180,E1 -31145.121,E2 -31145.121} C_VEL
LIN {X 0,Y 130.647,Z 512.924,A -85,B 0,C 180,E1 -31145.721,E2 -31145.721} C_VEL
LIN {X 0,Y 139.53,Z 499.163,A -85,B 0,C 180,E1 -31146.062,E2 -31146.062} C_VEL
LIN {X 0,Y 147.617,Z 484.016,A -85,B 0,C 180,E1 -31146.435,E2 -31146.435} C_VEL
LIN {X 0,Y 154.32,Z 468.713,A -85,B 0,C 180,E1 -31146.671,E2 -31146.671} C_VEL
LIN {X 0,Y 159.906,Z 452.683,A -85,B 0,C 180,E1 -31146.847,E2 -31146.847} C_VEL
LIN {X 0,Y 164.21,Z 436.303,A -85,B 0,C 180,E1 -31146.978,E2 -31146.978} C_VEL
LIN {X 0,Y 167.175,Z 419.686,A -85,B 0,C 180,E1 -31147.148,E2 -31147.148} C_VEL
LIN {X 0,Y 167.555,Z 416.894,A -85,B 0,C 180,E1 -31147.175,E2 -31147.175} C_VEL
LIN {X 0,Y 167.601,Z 415.899,A -85,B 0,C 180,E1 -31147.522,E2 -31147.522} C_VEL
LIN {X 0,Y 167.316,Z 415.956,A -85,B 0,C 180,E1 -31148.557,E2 -31148.557} C_VEL
LIN {X 0,Y 166.764,Z 417.312,A -85,B 0,C 180,E1 -31150.403,E2 -31150.403} C_VEL
LIN {X 0,Y 166.711,Z 417.252,A -85,B 0,C 180,E1 -31150.837,E2 -31150.837} C_VEL
LIN {X 0,Y 166.67,Z 416.627,A -85,B 0,C 180,E1 -31152.173,E2 -31152.173} C_VEL
LIN {X 0,Y 166.619,Z 416.791,A -85,B 0,C 180,E1 -31154.485,E2 -31154.485} C_VEL
LIN {X 0,Y 166.707,Z 418.48,A -85,B 0,C 180,E1 -31157.758,E2 -31157.758} C_VEL
LIN {X 0,Y 163.469,Z 436.487,A -85,B 0,C 180,E1 -31157.926,E2 -31157.926} C_VEL
LIN {X 0,Y 158.924,Z 453.357,A -85,B 0,C 180,E1 -31158.063,E2 -31158.063} C_VEL
LIN {X 0,Y 153.087,Z 469.657,A -85,B 0,C 180,E1 -31158.271,E2 -31158.271} C_VEL
LIN {X 0,Y 146.348,Z 484.656,A -85,B 0,C 180,E1 -31158.506,E2 -31158.506} C_VEL
LIN {X 0,Y 139.162,Z 498.032,A -85,B 0,C 180,E1 -31158.78,E2 -31158.78} C_VEL
LIN {X 0,Y 129.286,Z 513.291,A -85,B 0,C 180,E1 -31159.147,E2 -31159.147} C_VEL
LIN {X 0,Y 118.41,Z 527.298,A -85,B 0,C 180,E1 -31159.601,E2 -31159.601} C_VEL
LIN {X 0,Y 106.668,Z 540.075,A -85,B 0,C 180,E1 -31160.167,E2 -31160.167} C_VEL
LIN {X 0,Y 94.045,Z 551.749,A -85,B 0,C 180,E1 -31160.947,E2 -31160.947} C_VEL
LIN {X 0,Y 81.394,Z 561.726,A -85,B 0,C 180,E1 -31161.88,E2 -31161.88} C_VEL
LIN {X 0,Y 68.748,Z 570.262,A -85,B 0,C 180,E1 -31163.106,E2 -31163.106} C_VEL
LIN {X 0,Y 54.266,Z 578.435,A -85,B 0,C 180,E1 -31165.011,E2 -31165.011} C_VEL
LIN {X 0,Y 39.817,Z 585.185,A -85,B 0,C 180,E1 -31168.105,E2 -31168.105} C_VEL
LIN {X 0,Y 25.103,Z 590.787,A -85,B 0,C 180,E1 -31174.061,E2 -31174.061} C_VEL
LIN {X 0,Y 14.574,Z 594.019,A -85,B 0,C 180,E1 -31183.769,E2 -31183.769} C_VEL
LIN {X 0,Y 5.323,Z 596.739,A -85,B 0,C 180,E1 -31230.182,E2 -31230.182} C_VEL
LIN {X 0,Y 10.176,Z 598.791,A -85,B 0,C 180,E1 -31319.979,E2 -31319.979} C_VEL
LIN {X 0,Y 14.256,Z 599.404,A -85,B 0,C 180,E1 -31329.204,E2 -31329.204} C_VEL
LIN {X 0,Y 14.622,Z 599.496,A -85,B 0,C 180,E1 -31335.757,E2 -31335.757} C_VEL
LIN {X 0,Y 5.686,Z 597.585,A -85,B 0,C 180,E1 -31409.83,E2 -31409.83} C_VEL
LIN {X 0,Y 14.578,Z 594.399,A -85,B 0,C 180,E1 -31484.36,E2 -31484.36} C_VEL
LIN {X 0,Y 28.137,Z 590.104,A -85,B 0,C 180,E1 -31496.839,E2 -31496.839} C_VEL
LIN {X 0,Y 42.166,Z 584.607,A -85,B 0,C 180,E1 -31501.623,E2 -31501.623} C_VEL
LIN {X 0,Y 56.359,Z 577.735,A -85,B 0,C 180,E1 -31504.239,E2 -31504.239} C_VEL
LIN {X 0,Y 70.626,Z 569.448,A -85,B 0,C 180,E1 -31505.831,E2 -31505.831} C_VEL
LIN {X 0,Y 83.138,Z 560.901,A -85,B 0,C 180,E1 -31506.765,E2 -31506.765} C_VEL
LIN {X 0,Y 95.694,Z 550.74,A -85,B 0,C 180,E1 -31507.584,E2 -31507.584} C_VEL
LIN {X 0,Y 106.449,Z 540.699,A -85,B 0,C 180,E1 -31508.056,E2 -31508.056} C_VEL
LIN {X 0,Y 118.094,Z 528.094,A -85,B 0,C 180,E1 -31508.426,E2 -31508.426} C_VEL
LIN {X 0,Y 128.875,Z 514.275,A -85,B 0,C 180,E1 -31508.792,E2 -31508.792} C_VEL
LIN {X 0,Y 138.714,Z 499.194,A -85,B 0,C 180,E1 -31508.964,E2 -31508.964} C_VEL
LIN {X 0,Y 146.81,Z 484.151,A -85,B 0,C 180,E1 -31509.181,E2 -31509.181} C_VEL
LIN {X 0,Y 153.536,Z 468.939,A -85,B 0,C 180,E1 -31509.298,E2 -31509.298} C_VEL
LIN {X 0,Y 159.069,Z 453.286,A -85,B 0,C 180,E1 -31509.376,E2 -31509.376} C_VEL
LIN {X 0,Y 163.487,Z 436.77,A -85,B 0,C 180,E1 -31509.452,E2 -31509.452} C_VEL
LIN {X 0,Y 166.368,Z 420.997,A -85,B 0,C 180,E1 -31509.557,E2 -31509.557} C_VEL
LIN {X 0,Y 166.826,Z 417.863,A -85,B 0,C 180,E1 -31509.601,E2 -31509.601} C_VEL
LIN {X 0,Y 166.711,Z 417.252,A -85,B 0,C 180,E1 -31510.837,E2 -31510.837} C_VEL
LIN {X 0,Y 166.59,Z 417.461,A -85,B 0,C 180,E1 -31511.743,E2 -31511.743} C_VEL
LIN {X 0,Y 166.321,Z 418.972,A -85,B 0,C 180,E1 -31512.783,E2 -31512.783} C_VEL
LIN {X 0,Y 165.943,Z 421.341,A -85,B 0,C 180,E1 -31513.664,E2 -31513.664} C_VEL
LIN {X 0,Y 165.157,Z 426.405,A -85,B 0,C 180,E1 -31514.754,E2 -31514.754} C_VEL
LIN {X 0,Y 164.362,Z 430.698,A -85,B 0,C 180,E1 -31515.266,E2 -31515.266} C_VEL
LIN {X 0,Y 163.75,Z 433.674,A -85,B 0,C 180,E1 -31515.428,E2 -31515.428} C_VEL
LIN {X 0,Y 159.367,Z 450.898,A -85,B 0,C 180,E1 -31515.488,E2 -31515.488} C_VEL
LIN {X 0,Y 153.968,Z 466.707,A -85,B 0,C 180,E1 -31515.593,E2 -31515.593} C_VEL
LIN {X 0,Y 147.817,Z 481.123,A -85,B 0,C 180,E1 -31515.711,E2 -31515.711} C_VEL
LIN {X 0,Y 139.702,Z 496.548,A -85,B 0,C 180,E1 -31515.854,E2 -31515.854} C_VEL
LIN {X 0,Y 130.442,Z 511.141,A -85,B 0,C 180,E1 -31515.99,E2 -31515.99} C_VEL
LIN {X 0,Y 119.789,Z 525.227,A -85,B 0,C 180,E1 -31516.149,E2 -31516.149} C_VEL
LIN {X 0,Y 108.001,Z 538.376,A -85,B 0,C 180,E1 -31516.334,E2 -31516.334} C_VEL
LIN {X 0,Y 95.315,Z 550.361,A -85,B 0,C 180,E1 -31516.597,E2 -31516.597} C_VEL
LIN {X 0,Y 82.596,Z 560.602,A -85,B 0,C 180,E1 -31516.863,E2 -31516.863} C_VEL
LIN {X 0,Y 69.406,Z 569.552,A -85,B 0,C 180,E1 -31517.184,E2 -31517.184} C_VEL
LIN {X 0,Y 55.243,Z 577.66,A -85,B 0,C 180,E1 -31517.485,E2 -31517.485} C_VEL
LIN {X 0,Y 40.579,Z 584.62,A -85,B 0,C 180,E1 -31517.803,E2 -31517.803} C_VEL
LIN {X 0,Y 26.411,Z 590.056,A -85,B 0,C 180,E1 -31517.835,E2 -31517.835} C_VEL
LIN {X 0,Y 14.56,Z 593.724,A -85,B 0,C 180,E1 -31515.383,E2 -31515.383} C_VEL
LIN {X 0,Y 14.41,Z 593.777,A -85,B 0,C 180,E1 -31513.042,E2 -31513.042} C_VEL
LIN {X 0,Y 28.659,Z 589.316,A -85,B 0,C 180,E1 -31511.395,E2 -31511.395} C_VEL
LIN {X 0,Y 42.984,Z 583.692,A -85,B 0,C 180,E1 -31511.308,E2 -31511.308} C_VEL
LIN {X 0,Y 57.349,Z 576.681,A -85,B 0,C 180,E1 -31511.464,E2 -31511.464} C_VEL
LIN {X 0,Y 71.732,Z 568.187,A -85,B 0,C 180,E1 -31511.626,E2 -31511.626} C_VEL
LIN {X 0,Y 84.314,Z 559.417,A -85,B 0,C 180,E1 -31511.713,E2 -31511.713} C_VEL
LIN {X 0,Y 96.915,Z 549.142,A -85,B 0,C 180,E1 -31511.828,E2 -31511.828} C_VEL
LIN {X 0,Y 109.497,Z 537.003,A -85,B 0,C 180,E1 -31511.87,E2 -31511.87} C_VEL
LIN {X 0,Y 120.274,Z 524.79,A -85,B 0,C 180,E1 -31511.881,E2 -31511.881} C_VEL
LIN {X 0,Y 130.972,Z 510.514,A -85,B 0,C 180,E1 -31511.949,E2 -31511.949} C_VEL
LIN {X 0,Y 140.034,Z 496.112,A -85,B 0,C 180,E1 -31511.903,E2 -31511.903} C_VEL
LIN {X 0,Y 148.146,Z 480.54,A -85,B 0,C 180,E1 -31511.961,E2 -31511.961} C_VEL
LIN {X 0,Y 154.882,Z 464.553,A -85,B 0,C 180,E1 -31511.963,E2 -31511.963} C_VEL
LIN {X 0,Y 160.338,Z 447.801,A -85,B 0,C 180,E1 -31511.91,E2 -31511.91} C_VEL
